LIN {X 0,Y 254.112,Z 618.126,A -85,B 0,C 180,E1 -18637.149,E2 -18637.149} C_VEL
LIN {X 0,Y 253.777,Z 620.989,A -85,B 0,C 180,E1 -18639.564,E2 -18639.564} C_VEL
LIN {X 0,Y 253.688,Z 622.339,A -85,B 0,C 180,E1 -18641.181,E2 -18641.181} C_VEL
LIN {X 0,Y 253.728,Z 623.768,A -85,B 0,C 180,E1 -18644.196,E2 -18644.196} C_VEL
LIN {X 0,Y 253.789,Z 623.911,A -85,B 0,C 180,E1 -18646.076,E2 -18646.076} C_VEL
LIN {X 0,Y 253.947,Z 623.596,A -85,B 0,C 180,E1 -18647.723,E2 -18647.723} C_VEL
LIN {X 0,Y 254.457,Z 622.389,A -85,B 0,C 180,E1 -18650.104,E2 -18650.104} C_VEL
LIN {X 0,Y 255.585,Z 619.098,A -85,B 0,C 180,E1 -18653.497,E2 -18653.497} C_VEL
LIN {X 0,Y 256.833,Z 615.411,A -85,B 0,C 180,E1 -18655.964,E2 -18655.964} C_VEL
LIN {X 0,Y 258.431,Z 610.517,A -85,B 0,C 180,E1 -18658.418,E2 -18658.418} C_VEL
LIN {X 0,Y 260.518,Z 604.271,A -85,B 0,C 180,E1 -18660.834,E2 -18660.834} C_VEL
LIN {X 0,Y 262.965,Z 596.427,A -85,B 0,C 180,E1 -18663.221,E2 -18663.221} C_VEL
LIN {X 0,Y 265.473,Z 587.888,A -85,B 0,C 180,E1 -18665.261,E2 -18665.261} C_VEL
LIN {X 0,Y 268.117,Z 578.332,A -85,B 0,C 180,E1 -18667.076,E2 -18667.076} C_VEL
LIN {X 0,Y 270.488,Z 568.5,A -85,B 0,C 180,E1 -18668.577,E2 -18668.577} C_VEL
LIN {X 0,Y 272.671,Z 557.853,A -85,B 0,C 180,E1 -18669.877,E2 -18669.877} C_VEL
LIN {X 0,Y 274.602,Z 546.18,A -85,B 0,C 180,E1 -18670.981,E2 -18670.981} C_VEL
LIN {X 0,Y 276.337,Z 533.273,A -85,B 0,C 180,E1 -18671.853,E2 -18671.853} C_VEL
LIN {X 0,Y 277.554,Z 520.336,A -85,B 0,C 180,E1 -18672.432,E2 -18672.432} C_VEL
LIN {X 0,Y 280.067,Z 457.156,A -85,B 0,C 180,E1 -18674.084,E2 -18674.084} C_VEL
LIN {X 0,Y 274.463,Z 444.134,A -85,B 0,C 180,E1 -18675.366,E2 -18675.366} C_VEL
LIN {X 0,Y 267.207,Z 429.8,A -85,B 0,C 180,E1 -18677.057,E2 -18677.057} C_VEL
LIN {X 0,Y 260.209,Z 417.558,A -85,B 0,C 180,E1 -18678.762,E2 -18678.762} C_VEL
LIN {X 0,Y 257.879,Z 413.399,A -85,B 0,C 180,E1 -18679.453,E2 -18679.453} C_VEL
LIN {X 0,Y 256.173,Z 407.244,A -85,B 0,C 180,E1 -18682.71,E2 -18682.71} C_VEL
LIN {X 0,Y 256.081,Z 407.076,A -85,B 0,C 180,E1 -18686.709,E2 -18686.709} C_VEL
LIN {X 0,Y 256.122,Z 407.062,A -85,B 0,C 180,E1 -18691.409,E2 -18691.409} C_VEL
LIN {X 0,Y 256.162,Z 407.076,A -85,B 0,C 180,E1 -18695.699,E2 -18695.699} C_VEL
LIN {X 0,Y 256.162,Z 407.074,A -85,B 0,C 180,E1 -18699.105,E2 -18699.105} C_VEL
LIN {X 0,Y 256.289,Z 407.06,A -85,B 0,C 180,E1 -18704.084,E2 -18704.084} C_VEL
LIN {X 0,Y 256.304,Z 407.05,A -85,B 0,C 180,E1 -18708.934,E2 -18708.934} C_VEL
LIN {X 0,Y 256.533,Z 407.03,A -85,B 0,C 180,E1 -18712.127,E2 -18712.127} C_VEL
LIN {X 0,Y 256.347,Z 407.044,A -85,B 0,C 180,E1 -18715.171,E2 -18715.171} C_VEL
LIN {X 0,Y 255.716,Z 407.133,A -85,B 0,C 180,E1 -18716.486,E2 -18716.486} C_VEL
LIN {X 0,Y 253.085,Z 407.469,A -85,B 0,C 180,E1 -18718.637,E2 -18718.637} C_VEL
LIN {X 0,Y 249.973,Z 407.849,A -85,B 0,C 180,E1 -18721.28,E2 -18721.28} C_VEL
LIN {X 0,Y 249.565,Z 407.891,A -85,B 0,C 180,E1 -18722.191,E2 -18722.191} C_VEL
LIN {X 0,Y 249.455,Z 407.913,A -85,B 0,C 180,E1 -18726.471,E2 -18726.471} C_VEL
LIN {X 0,Y 249.383,Z 407.911,A -85,B 0,C 180,E1 -18729.735,E2 -18729.735} C_VEL
LIN {X 0,Y 249.199,Z 407.934,A -85,B 0,C 180,E1 -18734.704,E2 -18734.704} C_VEL
LIN {X 0,Y 249.134,Z 407.939,A -85,B 0,C 180,E1 -18738.078,E2 -18738.078} C_VEL
LIN {X 0,Y 249.082,Z 407.953,A -85,B 0,C 180,E1 -18741.519,E2 -18741.519} C_VEL
LIN {X 0,Y 249.126,Z 407.95,A -85,B 0,C 180,E1 -18745.483,E2 -18745.483} C_VEL
LIN {X 0,Y 249.079,Z 407.959,A -85,B 0,C 180,E1 -18748.994,E2 -18748.994} C_VEL
LIN {X 0,Y 249.032,Z 407.966,A -85,B 0,C 180,E1 -18752.426,E2 -18752.426} C_VEL
LIN {X 0,Y 249.072,Z 407.958,A -85,B 0,C 180,E1 -18756.339,E2 -18756.339} C_VEL
LIN {X 0,Y 249.082,Z 407.938,A -85,B 0,C 180,E1 -18760.463,E2 -18760.463} C_VEL
LIN {X 0,Y 249.017,Z 407.957,A -85,B 0,C 180,E1 -18764.876,E2 -18764.876} C_VEL
LIN {X 0,Y 249.039,Z 407.996,A -85,B 0,C 180,E1 -18766.648,E2 -18766.648} C_VEL
LIN {X 0,Y 250.574,Z 413.471,A -85,B 0,C 180,E1 -18769.829,E2 -18769.829} C_VEL
LIN {X 0,Y 252.023,Z 418.69,A -85,B 0,C 180,E1 -18772.439,E2 -18772.439} C_VEL
LIN {X 0,Y 254.643,Z 423.279,A -85,B 0,C 180,E1 -18773.215,E2 -18773.215} C_VEL
LIN {X 0,Y 263.1,Z 438.828,A -85,B 0,C 180,E1 -18775.383,E2 -18775.383} C_VEL
LIN {X 0,Y 270.526,Z 454.405,A -85,B 0,C 180,E1 -18777.189,E2 -18777.189} C_VEL
LIN {X 0,Y 272.23,Z 459.018,A -85,B 0,C 180,E1 -18777.618,E2 -18777.618} C_VEL
LIN {X 0,Y 273.963,Z 469.57,A -85,B 0,C 180,E1 -18778.237,E2 -18778.237} C_VEL
LIN {X 0,Y 271.409,Z 527.607,A -85,B 0,C 180,E1 -18779.779,E2 -18779.779} C_VEL
LIN {X 0,Y 270.097,Z 541.162,A -85,B 0,C 180,E1 -18780.425,E2 -18780.425} C_VEL
LIN {X 0,Y 268.197,Z 553.913,A -85,B 0,C 180,E1 -18781.324,E2 -18781.324} C_VEL
LIN {X 0,Y 265.918,Z 565.575,A -85,B 0,C 180,E1 -18782.452,E2 -18782.452} C_VEL
LIN {X 0,Y 263.435,Z 576.821,A -85,B 0,C 180,E1 -18783.885,E2 -18783.885} C_VEL
LIN {X 0,Y 260.778,Z 586.995,A -85,B 0,C 180,E1 -18785.522,E2 -18785.522} C_VEL
LIN {X 0,Y 257.805,Z 596.965,A -85,B 0,C 180,E1 -18787.565,E2 -18787.565} C_VEL
LIN {X 0,Y 255.094,Z 605.859,A -85,B 0,C 180,E1 -18789.894,E2 -18789.894} C_VEL
LIN {X 0,Y 252.844,Z 612.807,A -85,B 0,C 180,E1 -18792.197,E2 -18792.197} C_VEL
LIN {X 0,Y 250.801,Z 618.469,A -85,B 0,C 180,E1 -18794.562,E2 -18794.562} C_VEL
LIN {X 0,Y 249.326,Z 622.943,A -85,B 0,C 180,E1 -18796.968,E2 -18796.968} C_VEL
LIN {X 0,Y 248.525,Z 625.31,A -85,B 0,C 180,E1 -18798.583,E2 -18798.583} C_VEL
LIN {X 0,Y 247.412,Z 628.797,A -85,B 0,C 180,E1 -18801.835,E2 -18801.835} C_VEL
LIN {X 0,Y 246.945,Z 630.557,A -85,B 0,C 180,E1 -18804.937,E2 -18804.937} C_VEL
LIN {X 0,Y 246.831,Z 630.932,A -85,B 0,C 180,E1 -18806.736,E2 -18806.736} C_VEL
LIN {X 0,Y 246.859,Z 630.877,A -85,B 0,C 180,E1 -18808.369,E2 -18808.369} C_VEL
LIN {X 0,Y 246.899,Z 630.414,A -85,B 0,C 180,E1 -18810,E2 -18810} C_VEL
LIN {X 0,Y 246.86,Z 629.526,A -85,B 0,C 180,E1 -18811.632,E2 -18811.632} C_VEL
LIN {X 0,Y 246.831,Z 628.24,A -85,B 0,C 180,E1 -18813.265,E2 -18813.265} C_VEL
LIN {X 0,Y 246.906,Z 625.502,A -85,B 0,C 180,E1 -18815.718,E2 -18815.718} C_VEL
LIN {X 0,Y 247.269,Z 621.729,A -85,B 0,C 180,E1 -18818.17,E2 -18818.17} C_VEL
LIN {X 0,Y 247.852,Z 616.812,A -85,B 0,C 180,E1 -18820.621,E2 -18820.621} C_VEL
LIN {X 0,Y 248.729,Z 610.599,A -85,B 0,C 180,E1 -18823.064,E2 -18823.064} C_VEL
LIN {X 0,Y 250.11,Z 602.853,A -85,B 0,C 180,E1 -18825.483,E2 -18825.483} C_VEL
LIN {X 0,Y 251.484,Z 594.894,A -85,B 0,C 180,E1 -18827.483,E2 -18827.483} C_VEL
LIN {X 0,Y 252.89,Z 585.135,A -85,B 0,C 180,E1 -18829.481,E2 -18829.481} C_VEL
LIN {X 0,Y 254.533,Z 574.299,A -85,B 0,C 180,E1 -18831.248,E2 -18831.248} C_VEL
LIN {X 0,Y 256.086,Z 563.781,A -85,B 0,C 180,E1 -18832.595,E2 -18832.595} C_VEL
LIN {X 0,Y 257.649,Z 551.092,A -85,B 0,C 180,E1 -18833.831,E2 -18833.831} C_VEL
LIN {X 0,Y 258.828,Z 537.613,A -85,B 0,C 180,E1 -18834.782,E2 -18834.782} C_VEL
LIN {X 0,Y 259.618,Z 525.011,A -85,B 0,C 180,E1 -18835.344,E2 -18835.344} C_VEL
LIN {X 0,Y 261.246,Z 462.897,A -85,B 0,C 180,E1 -18837.047,E2 -18837.047} C_VEL
LIN {X 0,Y 257.5,Z 435.906,A -85,B 0,C 180,E1 -18838.198,E2 -18838.198} C_VEL
LIN {X 0,Y 251.549,Z 419.268,A -85,B 0,C 180,E1 -18839.345,E2 -18839.345} C_VEL
LIN {X 0,Y 249.312,Z 409.016,A -85,B 0,C 180,E1 -18843.345,E2 -18843.345} C_VEL
LIN {X 0,Y 249.092,Z 407.982,A -85,B 0,C 180,E1 -18843.925,E2 -18843.925} C_VEL
LIN {X 0,Y 249.043,Z 407.95,A -85,B 0,C 180,E1 -18848.377,E2 -18848.377} C_VEL
LIN {X 0,Y 249.044,Z 407.961,A -85,B 0,C 180,E1 -18852.801,E2 -18852.801} C_VEL
LIN {X 0,Y 249.062,Z 407.934,A -85,B 0,C 180,E1 -18857.372,E2 -18857.372} C_VEL
LIN {X 0,Y 249.052,Z 407.962,A -85,B 0,C 180,E1 -18861.624,E2 -18861.624} C_VEL
LIN {X 0,Y 249.061,Z 407.957,A -85,B 0,C 180,E1 -18865.642,E2 -18865.642} C_VEL
LIN {X 0,Y 249.046,Z 407.957,A -85,B 0,C 180,E1 -18869.472,E2 -18869.472} C_VEL
LIN {X 0,Y 249.067,Z 407.954,A -85,B 0,C 180,E1 -18873.161,E2 -18873.161} C_VEL
LIN {X 0,Y 249.059,Z 407.959,A -85,B 0,C 180,E1 -18876.73,E2 -18876.73} C_VEL
LIN {X 0,Y 249.105,Z 407.938,A -85,B 0,C 180,E1 -18880.211,E2 -18880.211} C_VEL
LIN {X 0,Y 249.24,Z 407.939,A -85,B 0,C 180,E1 -18883.622,E2 -18883.622} C_VEL
LIN {X 0,Y 249.241,Z 407.922,A -85,B 0,C 180,E1 -18888.616,E2 -18888.616} C_VEL
LIN {X 0,Y 249.452,Z 407.904,A -85,B 0,C 180,E1 -18891.902,E2 -18891.902} C_VEL
LIN {X 0,Y 249.294,Z 407.933,A -85,B 0,C 180,E1 -18895.148,E2 -18895.148} C_VEL
LIN {X 0,Y 249.673,Z 407.875,A -85,B 0,C 180,E1 -18898.387,E2 -18898.387} C_VEL
LIN {X 0,Y 249.673,Z 407.862,A -85,B 0,C 180,E1 -18901.613,E2 -18901.613} C_VEL
LIN {X 0,Y 249.438,Z 407.91,A -85,B 0,C 180,E1 -18906.711,E2 -18906.711} C_VEL
LIN {X 0,Y 249.341,Z 407.915,A -85,B 0,C 180,E1 -18909.736,E2 -18909.736} C_VEL
LIN {X 0,Y 249.198,Z 407.93,A -85,B 0,C 180,E1 -18914.704,E2 -18914.704} C_VEL
LIN {X 0,Y 249.136,Z 407.949,A -85,B 0,C 180,E1 -18918.077,E2 -18918.077} C_VEL
LIN {X 0,Y 249.085,Z 407.945,A -85,B 0,C 180,E1 -18921.518,E2 -18921.518} C_VEL
LIN {X 0,Y 249.128,Z 407.939,A -85,B 0,C 180,E1 -18925.482,E2 -18925.482} C_VEL
LIN {X 0,Y 249.081,Z 407.958,A -85,B 0,C 180,E1 -18928.993,E2 -18928.993} C_VEL
LIN {X 0,Y 249.028,Z 407.952,A -85,B 0,C 180,E1 -18932.426,E2 -18932.426} C_VEL
LIN {X 0,Y 249.046,Z 407.957,A -85,B 0,C 180,E1 -18936.343,E2 -18936.343} C_VEL
LIN {X 0,Y 249.004,Z 407.963,A -85,B 0,C 180,E1 -18940.478,E2 -18940.478} C_VEL
LIN {X 0,Y 249.009,Z 407.966,A -85,B 0,C 180,E1 -18944.878,E2 -18944.878} C_VEL
LIN {X 0,Y 249.036,Z 407.96,A -85,B 0,C 180,E1 -18947.368,E2 -18947.368} C_VEL
LIN {X 0,Y 249.051,Z 407.964,A -85,B 0,C 180,E1 -18951.624,E2 -18951.624} C_VEL
LIN {X 0,Y 249.061,Z 407.942,A -85,B 0,C 180,E1 -18955.643,E2 -18955.643} C_VEL
LIN {X 0,Y 249.052,Z 407.947,A -85,B 0,C 180,E1 -18959.473,E2 -18959.473} C_VEL
LIN {X 0,Y 249.074,Z 407.951,A -85,B 0,C 180,E1 -18963.162,E2 -18963.162} C_VEL
LIN {X 0,Y 249.08,Z 407.948,A -85,B 0,C 180,E1 -18966.733,E2 -18966.733} C_VEL
LIN {X 0,Y 249.196,Z 408.095,A -85,B 0,C 180,E1 -18971.555,E2 -18971.555} C_VEL
LIN {X 0,Y 250.291,Z 413.05,A -85,B 0,C 180,E1 -18973.576,E2 -18973.576} C_VEL
LIN {X 0,Y 256.255,Z 428.663,A -85,B 0,C 180,E1 -18974.719,E2 -18974.719} C_VEL
LIN {X 0,Y 259.336,Z 438.01,A -85,B 0,C 180,E1 -18975.295,E2 -18975.295} C_VEL
LIN {X 0,Y 261.649,Z 453.277,A -85,B 0,C 180,E1 -18975.961,E2 -18975.961} C_VEL
LIN {X 0,Y 259.555,Z 520.29,A -85,B 0,C 180,E1 -18977.787,E2 -18977.787} C_VEL
LIN {X 0,Y 258.768,Z 533.398,A -85,B 0,C 180,E1 -18978.445,E2 -18978.445} C_VEL
LIN {X 0,Y 257.68,Z 545.229,A -85,B 0,C 180,E1 -18979.316,E2 -18979.316} C_VEL
LIN {X 0,Y 256.248,Z 557.373,A -85,B 0,C 180,E1 -18980.528,E2 -18980.528} C_VEL
LIN {X 0,Y 254.517,Z 569.044,A -85,B 0,C 180,E1 -18982.064,E2 -18982.064} C_VEL
LIN {X 0,Y 253.082,Z 578.437,A -85,B 0,C 180,E1 -18983.622,E2 -18983.622} C_VEL
LIN {X 0,Y 251.443,Z 588.078,A -85,B 0,C 180,E1 -18985.591,E2 -18985.591} C_VEL
LIN {X 0,Y 250.22,Z 595.954,A -85,B 0,C 180,E1 -18987.585,E2 -18987.585} C_VEL
LIN {X 0,Y 248.882,Z 603.666,A -85,B 0,C 180,E1 -18990,E2 -18990} C_VEL
LIN {X 0,Y 247.955,Z 609.852,A -85,B 0,C 180,E1 -18992.436,E2 -18992.436} C_VEL
LIN {X 0,Y 247.399,Z 614.759,A -85,B 0,C 180,E1 -18994.888,E2 -18994.888} C_VEL
LIN {X 0,Y 246.973,Z 618.549,A -85,B 0,C 180,E1 -18997.357,E2 -18997.357} C_VEL
LIN {X 0,Y 246.675,Z 621.31,A -85,B 0,C 180,E1 -18999.842,E2 -18999.842} C_VEL
LIN {X 0,Y 246.598,Z 622.611,A -85,B 0,C 180,E1 -19001.507,E2 -19001.507} C_VEL
LIN {X 0,Y 246.648,Z 623.865,A -85,B 0,C 180,E1 -19004.35,E2 -19004.35} C_VEL
LIN {X 0,Y 246.737,Z 623.989,A -85,B 0,C 180,E1 -19006.548,E2 -19006.548} C_VEL
LIN {X 0,Y 246.954,Z 623.626,A -85,B 0,C 180,E1 -19008.242,E2 -19008.242} C_VEL
LIN {X 0,Y 247.432,Z 622.525,A -85,B 0,C 180,E1 -19010.393,E2 -19010.393} C_VEL
LIN {X 0,Y 248.394,Z 619.898,A -85,B 0,C 180,E1 -19013.334,E2 -19013.334} C_VEL
LIN {X 0,Y 249.537,Z 616.773,A -85,B 0,C 180,E1 -19015.677,E2 -19015.677} C_VEL
LIN {X 0,Y 251.248,Z 611.893,A -85,B 0,C 180,E1 -19018.393,E2 -19018.393} C_VEL
LIN {X 0,Y 253.528,Z 605.511,A -85,B 0,C 180,E1 -19021.049,E2 -19021.049} C_VEL
LIN {X 0,Y 255.822,Z 598.512,A -85,B 0,C 180,E1 -19023.328,E2 -19023.328} C_VEL
LIN {X 0,Y 258.479,Z 590.1,A -85,B 0,C 180,E1 -19025.502,E2 -19025.502} C_VEL
LIN {X 0,Y 261.351,Z 580.456,A -85,B 0,C 180,E1 -19027.473,E2 -19027.473} C_VEL
LIN {X 0,Y 264.095,Z 569.707,A -85,B 0,C 180,E1 -19029.198,E2 -19029.198} C_VEL
LIN {X 0,Y 266.618,Z 558.006,A -85,B 0,C 180,E1 -19030.672,E2 -19030.672} C_VEL
LIN {X 0,Y 268.715,Z 545.893,A -85,B 0,C 180,E1 -19031.829,E2 -19031.829} C_VEL
LIN {X 0,Y 270.575,Z 532.505,A -85,B 0,C 180,E1 -19032.731,E2 -19032.731} C_VEL
LIN {X 0,Y 271.77,Z 519.507,A -85,B 0,C 180,E1 -19033.307,E2 -19033.307} C_VEL
LIN {X 0,Y 274.325,Z 459.31,A -85,B 0,C 180,E1 -19034.892,E2 -19034.892} C_VEL
LIN {X 0,Y 268.112,Z 445.144,A -85,B 0,C 180,E1 -19036.376,E2 -19036.376} C_VEL
LIN {X 0,Y 260.809,Z 430.871,A -85,B 0,C 180,E1 -19038.169,E2 -19038.169} C_VEL
LIN {X 0,Y 253.015,Z 417.7,A -85,B 0,C 180,E1 -19040.177,E2 -19040.177} C_VEL
LIN {X 0,Y 250.681,Z 413.682,A -85,B 0,C 180,E1 -19040.891,E2 -19040.891} C_VEL
LIN {X 0,Y 249.687,Z 410.098,A -85,B 0,C 180,E1 -19042.759,E2 -19042.759} C_VEL
LIN {X 0,Y 249.091,Z 407.978,A -85,B 0,C 180,E1 -19044.145,E2 -19044.145} C_VEL
LIN {X 0,Y 249.035,Z 407.965,A -85,B 0,C 180,E1 -19047.844,E2 -19047.844} C_VEL
LIN {X 0,Y 249.081,Z 407.938,A -85,B 0,C 180,E1 -19051.336,E2 -19051.336} C_VEL
LIN {X 0,Y 249.147,Z 407.945,A -85,B 0,C 180,E1 -19054.968,E2 -19054.968} C_VEL
LIN {X 0,Y 249.106,Z 407.955,A -85,B 0,C 180,E1 -19060.211,E2 -19060.211} C_VEL
LIN {X 0,Y 249.236,Z 407.939,A -85,B 0,C 180,E1 -19063.622,E2 -19063.622} C_VEL
LIN {X 0,Y 249.247,Z 407.932,A -85,B 0,C 180,E1 -19068.616,E2 -19068.616} C_VEL
LIN {X 0,Y 249.475,Z 407.909,A -85,B 0,C 180,E1 -19071.903,E2 -19071.903} C_VEL
LIN {X 0,Y 249.462,Z 407.913,A -85,B 0,C 180,E1 -19076.77,E2 -19076.77} C_VEL
LIN {X 0,Y 249.73,Z 407.868,A -85,B 0,C 180,E1 -19080,E2 -19080} C_VEL
LIN {X 0,Y 249.565,Z 407.891,A -85,B 0,C 180,E1 -19082.191,E2 -19082.191} C_VEL
LIN {X 0,Y 248.748,Z 407.989,A -85,B 0,C 180,E1 -19083.537,E2 -19083.537} C_VEL
LIN {X 0,Y 245.844,Z 408.361,A -85,B 0,C 180,E1 -19085.733,E2 -19085.733} C_VEL
LIN {X 0,Y 243.465,Z 408.652,A -85,B 0,C 180,E1 -19087.521,E2 -19087.521} C_VEL
LIN {X 0,Y 242.448,Z 408.771,A -85,B 0,C 180,E1 -19088.907,E2 -19088.907} C_VEL
LIN {X 0,Y 242.362,Z 408.783,A -85,B 0,C 180,E1 -19089.377,E2 -19089.377} C_VEL
LIN {X 0,Y 242.161,Z 408.815,A -85,B 0,C 180,E1 -19095.141,E2 -19095.141} C_VEL
LIN {X 0,Y 242.068,Z 408.819,A -85,B 0,C 180,E1 -19098.625,E2 -19098.625} C_VEL
LIN {X 0,Y 242.008,Z 408.829,A -85,B 0,C 180,E1 -19102.181,E2 -19102.181} C_VEL
LIN {X 0,Y 242.062,Z 408.826,A -85,B 0,C 180,E1 -19105.839,E2 -19105.839} C_VEL
LIN {X 0,Y 242.026,Z 408.834,A -85,B 0,C 180,E1 -19109.581,E2 -19109.581} C_VEL
LIN {X 0,Y 241.987,Z 408.836,A -85,B 0,C 180,E1 -19113.492,E2 -19113.492} C_VEL
LIN {X 0,Y 242.016,Z 408.832,A -85,B 0,C 180,E1 -19117.577,E2 -19117.577} C_VEL
LIN {X 0,Y 241.984,Z 408.817,A -85,B 0,C 180,E1 -19121.913,E2 -19121.913} C_VEL
LIN {X 0,Y 241.995,Z 409.041,A -85,B 0,C 180,E1 -19125.45,E2 -19125.45} C_VEL
LIN {X 0,Y 244.075,Z 416.279,A -85,B 0,C 180,E1 -19129.717,E2 -19129.717} C_VEL
LIN {X 0,Y 244.789,Z 418.663,A -85,B 0,C 180,E1 -19130.877,E2 -19130.877} C_VEL
LIN {X 0,Y 247.405,Z 423.195,A -85,B 0,C 180,E1 -19131.703,E2 -19131.703} C_VEL
LIN {X 0,Y 253.58,Z 434.009,A -85,B 0,C 180,E1 -19133.406,E2 -19133.406} C_VEL
LIN {X 0,Y 259.89,Z 446.068,A -85,B 0,C 180,E1 -19135.057,E2 -19135.057} C_VEL
LIN {X 0,Y 266.039,Z 459.536,A -85,B 0,C 180,E1 -19136.615,E2 -19136.615} C_VEL
LIN {X 0,Y 266.95,Z 462.519,A -85,B 0,C 180,E1 -19136.87,E2 -19136.87} C_VEL
LIN {X 0,Y 268.284,Z 470.283,A -85,B 0,C 180,E1 -19137.354,E2 -19137.354} C_VEL
LIN {X 0,Y 265.717,Z 526.862,A -85,B 0,C 180,E1 -19138.878,E2 -19138.878} C_VEL
LIN {X 0,Y 264.317,Z 540.529,A -85,B 0,C 180,E1 -19139.52,E2 -19139.52} C_VEL
LIN {X 0,Y 262.427,Z 553.183,A -85,B 0,C 180,E1 -19140.412,E2 -19140.412} C_VEL
LIN {X 0,Y 260.04,Z 564.991,A -85,B 0,C 180,E1 -19141.554,E2 -19141.554} C_VEL
LIN {X 0,Y 257.463,Z 576.317,A -85,B 0,C 180,E1 -19143.012,E2 -19143.012} C_VEL
LIN {X 0,Y 254.697,Z 586.561,A -85,B 0,C 180,E1 -19144.679,E2 -19144.679} C_VEL
LIN {X 0,Y 251.817,Z 595.795,A -85,B 0,C 180,E1 -19146.566,E2 -19146.566} C_VEL
LIN {X 0,Y 249.014,Z 604.498,A -85,B 0,C 180,E1 -19148.831,E2 -19148.831} C_VEL
LIN {X 0,Y 246.517,Z 611.976,A -85,B 0,C 180,E1 -19151.294,E2 -19151.294} C_VEL
LIN {X 0,Y 244.613,Z 616.899,A -85,B 0,C 180,E1 -19153.304,E2 -19153.304} C_VEL
LIN {X 0,Y 242.857,Z 621.69,A -85,B 0,C 180,E1 -19155.761,E2 -19155.761} C_VEL
LIN {X 0,Y 241.554,Z 625.386,A -85,B 0,C 180,E1 -19158.249,E2 -19158.249} C_VEL
LIN {X 0,Y 240.891,Z 627.303,A -85,B 0,C 180,E1 -19159.919,E2 -19159.919} C_VEL
LIN {X 0,Y 240.386,Z 628.805,A -85,B 0,C 180,E1 -19161.595,E2 -19161.595} C_VEL
LIN {X 0,Y 239.845,Z 630.545,A -85,B 0,C 180,E1 -19164.957,E2 -19164.957} C_VEL
LIN {X 0,Y 239.773,Z 630.76,A -85,B 0,C 180,E1 -19168.321,E2 -19168.321} C_VEL
LIN {X 0,Y 239.811,Z 630.247,A -85,B 0,C 180,E1 -19170,E2 -19170} C_VEL
LIN {X 0,Y 239.774,Z 629.332,A -85,B 0,C 180,E1 -19171.68,E2 -19171.68} C_VEL
LIN {X 0,Y 239.766,Z 626.645,A -85,B 0,C 180,E1 -19174.718,E2 -19174.718} C_VEL
LIN {X 0,Y 240.048,Z 622.813,A -85,B 0,C 180,E1 -19177.571,E2 -19177.571} C_VEL
LIN {X 0,Y 240.618,Z 618.229,A -85,B 0,C 180,E1 -19180.093,E2 -19180.093} C_VEL
LIN {X 0,Y 241.584,Z 611.251,A -85,B 0,C 180,E1 -19183.03,E2 -19183.03} C_VEL
LIN {X 0,Y 242.966,Z 603.689,A -85,B 0,C 180,E1 -19185.519,E2 -19185.519} C_VEL
LIN {X 0,Y 244.362,Z 595.951,A -85,B 0,C 180,E1 -19187.577,E2 -19187.577} C_VEL
LIN {X 0,Y 245.888,Z 586.075,A -85,B 0,C 180,E1 -19189.705,E2 -19189.705} C_VEL
LIN {X 0,Y 247.671,Z 574.634,A -85,B 0,C 180,E1 -19191.647,E2 -19191.647} C_VEL
LIN {X 0,Y 249.272,Z 564.232,A -85,B 0,C 180,E1 -19193.029,E2 -19193.029} C_VEL
LIN {X 0,Y 250.871,Z 551.751,A -85,B 0,C 180,E1 -19194.297,E2 -19194.297} C_VEL
LIN {X 0,Y 252.104,Z 538.553,A -85,B 0,C 180,E1 -19195.269,E2 -19195.269} C_VEL
LIN {X 0,Y 252.968,Z 525.413,A -85,B 0,C 180,E1 -19195.893,E2 -19195.893} C_VEL
LIN {X 0,Y 254.789,Z 464.792,A -85,B 0,C 180,E1 -19197.584,E2 -19197.584} C_VEL
LIN {X 0,Y 251.148,Z 438.097,A -85,B 0,C 180,E1 -19198.758,E2 -19198.758} C_VEL
LIN {X 0,Y 245.146,Z 421.605,A -85,B 0,C 180,E1 -19199.902,E2 -19199.902} C_VEL
LIN {X 0,Y 244.224,Z 418.953,A -85,B 0,C 180,E1 -19200.175,E2 -19200.175} C_VEL
LIN {X 0,Y 242.201,Z 409.661,A -85,B 0,C 180,E1 -19203.957,E2 -19203.957} C_VEL
LIN {X 0,Y 242.042,Z 408.85,A -85,B 0,C 180,E1 -19204.486,E2 -19204.486} C_VEL
LIN {X 0,Y 242.011,Z 408.825,A -85,B 0,C 180,E1 -19208.364,E2 -19208.364} C_VEL
LIN {X 0,Y 241.966,Z 408.845,A -85,B 0,C 180,E1 -19211.916,E2 -19211.916} C_VEL
LIN {X 0,Y 241.991,Z 408.807,A -85,B 0,C 180,E1 -19216.557,E2 -19216.557} C_VEL
LIN {X 0,Y 242.008,Z 408.839,A -85,B 0,C 180,E1 -19220.291,E2 -19220.291} C_VEL
LIN {X 0,Y 242.036,Z 408.825,A -85,B 0,C 180,E1 -19224.497,E2 -19224.497} C_VEL
LIN {X 0,Y 241.973,Z 408.843,A -85,B 0,C 180,E1 -19228.479,E2 -19228.479} C_VEL
LIN {X 0,Y 241.999,Z 408.831,A -85,B 0,C 180,E1 -19232.311,E2 -19232.311} C_VEL
LIN {X 0,Y 242.039,Z 408.834,A -85,B 0,C 180,E1 -19236.014,E2 -19236.014} C_VEL
LIN {X 0,Y 242.033,Z 408.817,A -85,B 0,C 180,E1 -19239.607,E2 -19239.607} C_VEL
LIN {X 0,Y 242.161,Z 408.818,A -85,B 0,C 180,E1 -19243.278,E2 -19243.278} C_VEL
LIN {X 0,Y 242.178,Z 408.803,A -85,B 0,C 180,E1 -19248.279,E2 -19248.279} C_VEL
LIN {X 0,Y 242.398,Z 408.778,A -85,B 0,C 180,E1 -19251.664,E2 -19251.664} C_VEL
LIN {X 0,Y 242.255,Z 408.809,A -85,B 0,C 180,E1 -19255.007,E2 -19255.007} C_VEL
LIN {X 0,Y 242.633,Z 408.752,A -85,B 0,C 180,E1 -19258.34,E2 -19258.34} C_VEL
LIN {X 0,Y 242.633,Z 408.738,A -85,B 0,C 180,E1 -19261.66,E2 -19261.66} C_VEL
LIN {X 0,Y 242.419,Z 408.787,A -85,B 0,C 180,E1 -19266.683,E2 -19266.683} C_VEL
LIN {X 0,Y 242.265,Z 408.795,A -85,B 0,C 180,E1 -19270.024,E2 -19270.024} C_VEL
LIN {X 0,Y 242.161,Z 408.809,A -85,B 0,C 180,E1 -19275.141,E2 -19275.141} C_VEL
LIN {X 0,Y 242.07,Z 408.83,A -85,B 0,C 180,E1 -19278.624,E2 -19278.624} C_VEL
LIN {X 0,Y 242.011,Z 408.824,A -85,B 0,C 180,E1 -19282.18,E2 -19282.18} C_VEL
LIN {X 0,Y 242.065,Z 408.822,A -85,B 0,C 180,E1 -19285.838,E2 -19285.838} C_VEL
LIN {X 0,Y 242.028,Z 408.834,A -85,B 0,C 180,E1 -19289.58,E2 -19289.58} C_VEL
LIN {X 0,Y 241.979,Z 408.823,A -85,B 0,C 180,E1 -19293.493,E2 -19293.493} C_VEL
LIN {X 0,Y 241.987,Z 408.842,A -85,B 0,C 180,E1 -19297.582,E2 -19297.582} C_VEL
LIN {X 0,Y 241.938,Z 408.83,A -85,B 0,C 180,E1 -19301.922,E2 -19301.922} C_VEL
LIN {X 0,Y 241.973,Z 408.844,A -85,B 0,C 180,E1 -19306.561,E2 -19306.561} C_VEL
LIN {X 0,Y 241.987,Z 408.837,A -85,B 0,C 180,E1 -19310.287,E2 -19310.287} C_VEL
LIN {X 0,Y 242.037,Z 408.826,A -85,B 0,C 180,E1 -19314.498,E2 -19314.498} C_VEL
LIN {X 0,Y 241.976,Z 408.814,A -85,B 0,C 180,E1 -19318.48,E2 -19318.48} C_VEL
LIN {X 0,Y 242.01,Z 408.839,A -85,B 0,C 180,E1 -19322.313,E2 -19322.313} C_VEL
LIN {X 0,Y 242.058,Z 408.812,A -85,B 0,C 180,E1 -19326.016,E2 -19326.016} C_VEL
LIN {X 0,Y 242.174,Z 408.986,A -85,B 0,C 180,E1 -19331.055,E2 -19331.055} C_VEL
LIN {X 0,Y 243.104,Z 413.283,A -85,B 0,C 180,E1 -19332.812,E2 -19332.812} C_VEL
LIN {X 0,Y 249.796,Z 430.382,A -85,B 0,C 180,E1 -19334.12,E2 -19334.12} C_VEL
LIN {X 0,Y 253.035,Z 440.431,A -85,B 0,C 180,E1 -19334.758,E2 -19334.758} C_VEL
LIN {X 0,Y 255.082,Z 454.542,A -85,B 0,C 180,E1 -19335.388,E2 -19335.388} C_VEL
LIN {X 0,Y 252.96,Z 520.007,A -85,B 0,C 180,E1 -19337.209,E2 -19337.209} C_VEL
LIN {X 0,Y 252.117,Z 533.257,A -85,B 0,C 180,E1 -19337.881,E2 -19337.881} C_VEL
LIN {X 0,Y 250.877,Z 546.548,A -85,B 0,C 180,E1 -19338.895,E2 -19338.895} C_VEL
LIN {X 0,Y 249.469,Z 557.738,A -85,B 0,C 180,E1 -19340.063,E2 -19340.063} C_VEL
LIN {X 0,Y 247.68,Z 569.362,A -85,B 0,C 180,E1 -19341.638,E2 -19341.638} C_VEL
LIN {X 0,Y 246.199,Z 578.717,A -85,B 0,C 180,E1 -19343.237,E2 -19343.237} C_VEL
LIN {X 0,Y 244.675,Z 587.432,A -85,B 0,C 180,E1 -19345.056,E2 -19345.056} C_VEL
LIN {X 0,Y 243.355,Z 595.435,A -85,B 0,C 180,E1 -19347.103,E2 -19347.103} C_VEL
LIN {X 0,Y 241.931,Z 603.301,A -85,B 0,C 180,E1 -19349.583,E2 -19349.583} C_VEL
LIN {X 0,Y 241.163,Z 608.631,A -85,B 0,C 180,E1 -19351.67,E2 -19351.67} C_VEL
LIN {X 0,Y 240.45,Z 613.833,A -85,B 0,C 180,E1 -19354.19,E2 -19354.19} C_VEL
LIN {X 0,Y 239.989,Z 617.877,A -85,B 0,C 180,E1 -19356.726,E2 -19356.726} C_VEL
LIN {X 0,Y 239.691,Z 619.967,A -85,B 0,C 180,E1 -19358.43,E2 -19358.43} C_VEL
LIN {X 0,Y 239.546,Z 621.628,A -85,B 0,C 180,E1 -19360.138,E2 -19360.138} C_VEL
LIN {X 0,Y 239.49,Z 622.881,A -85,B 0,C 180,E1 -19361.853,E2 -19361.853} C_VEL
LIN {X 0,Y 239.552,Z 623.957,A -85,B 0,C 180,E1 -19364.498,E2 -19364.498} C_VEL
LIN {X 0,Y 239.688,Z 624.068,A -85,B 0,C 180,E1 -19367.05,E2 -19367.05} C_VEL
LIN {X 0,Y 239.957,Z 623.65,A -85,B 0,C 180,E1 -19368.794,E2 -19368.794} C_VEL
LIN {X 0,Y 240.41,Z 622.662,A -85,B 0,C 180,E1 -19370.696,E2 -19370.696} C_VEL
LIN {X 0,Y 241.569,Z 619.727,A -85,B 0,C 180,E1 -19374.035,E2 -19374.035} C_VEL
LIN {X 0,Y 242.988,Z 616.08,A -85,B 0,C 180,E1 -19376.715,E2 -19376.715} C_VEL
LIN {X 0,Y 244.73,Z 611.486,A -85,B 0,C 180,E1 -19379.221,E2 -19379.221} C_VEL
LIN {X 0,Y 247.01,Z 605.344,A -85,B 0,C 180,E1 -19381.791,E2 -19381.791} C_VEL
LIN {X 0,Y 249.645,Z 597.789,A -85,B 0,C 180,E1 -19384.265,E2 -19384.265} C_VEL
LIN {X 0,Y 252.172,Z 590.124,A -85,B 0,C 180,E1 -19386.264,E2 -19386.264} C_VEL
LIN {X 0,Y 255.211,Z 580.388,A -85,B 0,C 180,E1 -19388.286,E2 -19388.286} C_VEL
LIN {X 0,Y 257.96,Z 570,A -85,B 0,C 180,E1 -19389.988,E2 -19389.988} C_VEL
LIN {X 0,Y 260.409,Z 559.176,A -85,B 0,C 180,E1 -19391.391,E2 -19391.391} C_VEL
LIN {X 0,Y 262.693,Z 546.815,A -85,B 0,C 180,E1 -19392.624,E2 -19392.624} C_VEL
LIN {X 0,Y 264.611,Z 533.714,A -85,B 0,C 180,E1 -19393.541,E2 -19393.541} C_VEL
LIN {X 0,Y 265.98,Z 520.085,A -85,B 0,C 180,E1 -19394.169,E2 -19394.169} C_VEL
LIN {X 0,Y 268.618,Z 461.507,A -85,B 0,C 180,E1 -19395.738,E2 -19395.738} C_VEL
LIN {X 0,Y 263.095,Z 448.806,A -85,B 0,C 180,E1 -19397.119,E2 -19397.119} C_VEL
LIN {X 0,Y 256.329,Z 435.467,A -85,B 0,C 180,E1 -19398.85,E2 -19398.85} C_VEL
LIN {X 0,Y 250.496,Z 425.435,A -85,B 0,C 180,E1 -19400.401,E2 -19400.401} C_VEL
LIN {X 0,Y 245.604,Z 417.54,A -85,B 0,C 180,E1 -19401.775,E2 -19401.775} C_VEL
LIN {X 0,Y 243.39,Z 413.605,A -85,B 0,C 180,E1 -19402.555,E2 -19402.555} C_VEL
LIN {X 0,Y 242.059,Z 409.069,A -85,B 0,C 180,E1 -19405.264,E2 -19405.264} C_VEL
LIN {X 0,Y 241.991,Z 408.84,A -85,B 0,C 180,E1 -19407.374,E2 -19407.374} C_VEL
LIN {X 0,Y 242.009,Z 408.813,A -85,B 0,C 180,E1 -19410.596,E2 -19410.596} C_VEL
LIN {X 0,Y 242.063,Z 408.828,A -85,B 0,C 180,E1 -19414.183,E2 -19414.183} C_VEL
LIN {X 0,Y 242.048,Z 408.826,A -85,B 0,C 180,E1 -19418.297,E2 -19418.297} C_VEL
LIN {X 0,Y 242.158,Z 408.822,A -85,B 0,C 180,E1 -19423.278,E2 -19423.278} C_VEL
LIN {X 0,Y 242.18,Z 408.816,A -85,B 0,C 180,E1 -19428.28,E2 -19428.28} C_VEL
LIN {X 0,Y 242.422,Z 408.788,A -85,B 0,C 180,E1 -19431.666,E2 -19431.666} C_VEL
LIN {X 0,Y 242.263,Z 408.796,A -85,B 0,C 180,E1 -19435.007,E2 -19435.007} C_VEL
LIN {X 0,Y 242.641,Z 408.749,A -85,B 0,C 180,E1 -19438.34,E2 -19438.34} C_VEL
LIN {X 0,Y 242.633,Z 408.762,A -85,B 0,C 180,E1 -19441.66,E2 -19441.66} C_VEL
LIN {X 0,Y 242.427,Z 408.788,A -85,B 0,C 180,E1 -19446.659,E2 -19446.659} C_VEL
LIN {X 0,Y 242.362,Z 408.783,A -85,B 0,C 180,E1 -19449.377,E2 -19449.377} C_VEL
LIN {X 0,Y 241.656,Z 408.882,A -85,B 0,C 180,E1 -19450.762,E2 -19450.762} C_VEL
LIN {X 0,Y 238.698,Z 409.249,A -85,B 0,C 180,E1 -19453.017,E2 -19453.017} C_VEL
LIN {X 0,Y 236.207,Z 409.558,A -85,B 0,C 180,E1 -19454.856,E2 -19454.856} C_VEL
LIN {X 0,Y 235.16,Z 409.694,A -85,B 0,C 180,E1 -19456.285,E2 -19456.285} C_VEL
LIN {X 0,Y 235.086,Z 409.696,A -85,B 0,C 180,E1 -19456.77,E2 -19456.77} C_VEL
LIN {X 0,Y 235.007,Z 409.709,A -85,B 0,C 180,E1 -19461.031,E2 -19461.031} C_VEL
LIN {X 0,Y 234.99,Z 409.704,A -85,B 0,C 180,E1 -19466.207,E2 -19466.207} C_VEL
LIN {X 0,Y 234.928,Z 409.712,A -85,B 0,C 180,E1 -19470.568,E2 -19470.568} C_VEL
LIN {X 0,Y 234.957,Z 409.711,A -85,B 0,C 180,E1 -19474.634,E2 -19474.634} C_VEL
LIN {X 0,Y 234.965,Z 409.718,A -85,B 0,C 180,E1 -19478.953,E2 -19478.953} C_VEL
LIN {X 0,Y 234.964,Z 409.738,A -85,B 0,C 180,E1 -19483.719,E2 -19483.719} C_VEL
LIN {X 0,Y 235.697,Z 412.584,A -85,B 0,C 180,E1 -19485.695,E2 -19485.695} C_VEL
LIN {X 0,Y 237.435,Z 418.434,A -85,B 0,C 180,E1 -19489.096,E2 -19489.096} C_VEL
LIN {X 0,Y 240.196,Z 423.06,A -85,B 0,C 180,E1 -19490.039,E2 -19490.039} C_VEL
LIN {X 0,Y 246.49,Z 433.625,A -85,B 0,C 180,E1 -19491.917,E2 -19491.917} C_VEL
LIN {X 0,Y 254.631,Z 448.998,A -85,B 0,C 180,E1 -19494.172,E2 -19494.172} C_VEL
LIN {X 0,Y 260.946,Z 463.001,A -85,B 0,C 180,E1 -19495.85,E2 -19495.85} C_VEL
LIN {X 0,Y 261.853,Z 466.527,A -85,B 0,C 180,E1 -19496.134,E2 -19496.134} C_VEL
LIN {X 0,Y 262.605,Z 472.096,A -85,B 0,C 180,E1 -19496.459,E2 -19496.459} C_VEL
LIN {X 0,Y 260.014,Z 526.796,A -85,B 0,C 180,E1 -19497.96,E2 -19497.96} C_VEL
LIN {X 0,Y 258.556,Z 540.431,A -85,B 0,C 180,E1 -19498.608,E2 -19498.608} C_VEL
LIN {X 0,Y 256.727,Z 552.403,A -85,B 0,C 180,E1 -19499.46,E2 -19499.46} C_VEL
LIN {X 0,Y 254.227,Z 564.409,A -85,B 0,C 180,E1 -19500.615,E2 -19500.615} C_VEL
LIN {X 0,Y 251.551,Z 575.821,A -85,B 0,C 180,E1 -19502.098,E2 -19502.098} C_VEL
LIN {X 0,Y 248.61,Z 586.138,A -85,B 0,C 180,E1 -19503.788,E2 -19503.788} C_VEL
LIN {X 0,Y 245.918,Z 594.588,A -85,B 0,C 180,E1 -19505.52,E2 -19505.52} C_VEL
LIN {X 0,Y 242.889,Z 603.478,A -85,B 0,C 180,E1 -19507.808,E2 -19507.808} C_VEL
LIN {X 0,Y 240.239,Z 611.149,A -85,B 0,C 180,E1 -19510.342,E2 -19510.342} C_VEL
LIN {X 0,Y 237.807,Z 617.107,A -85,B 0,C 180,E1 -19512.811,E2 -19512.811} C_VEL
LIN {X 0,Y 235.947,Z 621.831,A -85,B 0,C 180,E1 -19515.335,E2 -19515.335} C_VEL
LIN {X 0,Y 234.58,Z 625.464,A -85,B 0,C 180,E1 -19517.895,E2 -19517.895} C_VEL
LIN {X 0,Y 233.875,Z 627.351,A -85,B 0,C 180,E1 -19519.613,E2 -19519.613} C_VEL
LIN {X 0,Y 233.354,Z 628.8,A -85,B 0,C 180,E1 -19521.34,E2 -19521.34} C_VEL
LIN {X 0,Y 232.769,Z 630.485,A -85,B 0,C 180,E1 -19524.804,E2 -19524.804} C_VEL
LIN {X 0,Y 232.656,Z 630.757,A -85,B 0,C 180,E1 -19526.537,E2 -19526.537} C_VEL
LIN {X 0,Y 232.67,Z 630.63,A -85,B 0,C 180,E1 -19528.27,E2 -19528.27} C_VEL
LIN {X 0,Y 232.725,Z 630.08,A -85,B 0,C 180,E1 -19530,E2 -19530} C_VEL
LIN {X 0,Y 232.67,Z 629.138,A -85,B 0,C 180,E1 -19531.731,E2 -19531.731} C_VEL
LIN {X 0,Y 232.679,Z 626.652,A -85,B 0,C 180,E1 -19534.614,E2 -19534.614} C_VEL
LIN {X 0,Y 233.004,Z 622.487,A -85,B 0,C 180,E1 -19537.801,E2 -19537.801} C_VEL
LIN {X 0,Y 233.588,Z 617.832,A -85,B 0,C 180,E1 -19540.4,E2 -19540.4} C_VEL
LIN {X 0,Y 234.642,Z 610.776,A -85,B 0,C 180,E1 -19543.423,E2 -19543.423} C_VEL
LIN {X 0,Y 236.101,Z 603.133,A -85,B 0,C 180,E1 -19545.983,E2 -19545.983} C_VEL
LIN {X 0,Y 237.569,Z 595.291,A -85,B 0,C 180,E1 -19548.097,E2 -19548.097} C_VEL
LIN {X 0,Y 239.113,Z 585.535,A -85,B 0,C 180,E1 -19550.229,E2 -19550.229} C_VEL
LIN {X 0,Y 240.822,Z 574.97,A -85,B 0,C 180,E1 -19552.07,E2 -19552.07} C_VEL
LIN {X 0,Y 242.718,Z 563.001,A -85,B 0,C 180,E1 -19553.688,E2 -19553.688} C_VEL
LIN {X 0,Y 244.386,Z 550.137,A -85,B 0,C 180,E1 -19554.985,E2 -19554.985} C_VEL
LIN {X 0,Y 245.605,Z 537.148,A -85,B 0,C 180,E1 -19555.93,E2 -19555.93} C_VEL
LIN {X 0,Y 246.404,Z 524.305,A -85,B 0,C 180,E1 -19556.523,E2 -19556.523} C_VEL
LIN {X 0,Y 248.148,Z 464.519,A -85,B 0,C 180,E1 -19558.237,E2 -19558.237} C_VEL
LIN {X 0,Y 244.821,Z 440.092,A -85,B 0,C 180,E1 -19559.348,E2 -19559.348} C_VEL
LIN {X 0,Y 239.006,Z 424.215,A -85,B 0,C 180,E1 -19560.498,E2 -19560.498} C_VEL
LIN {X 0,Y 236.972,Z 419.024,A -85,B 0,C 180,E1 -19560.969,E2 -19560.969} C_VEL
LIN {X 0,Y 235.736,Z 413.038,A -85,B 0,C 180,E1 -19563.408,E2 -19563.408} C_VEL
LIN {X 0,Y 235.004,Z 409.74,A -85,B 0,C 180,E1 -19564.976,E2 -19564.976} C_VEL
LIN {X 0,Y 234.942,Z 409.703,A -85,B 0,C 180,E1 -19568.944,E2 -19568.944} C_VEL
LIN {X 0,Y 234.958,Z 409.705,A -85,B 0,C 180,E1 -19573.469,E2 -19573.469} C_VEL
LIN {X 0,Y 234.964,Z 409.679,A -85,B 0,C 180,E1 -19576.532,E2 -19576.532} C_VEL
LIN {X 0,Y 234.955,Z 409.719,A -85,B 0,C 180,E1 -19581.086,E2 -19581.086} C_VEL
LIN {X 0,Y 234.96,Z 409.71,A -85,B 0,C 180,E1 -19585.367,E2 -19585.367} C_VEL
LIN {X 0,Y 234.922,Z 409.716,A -85,B 0,C 180,E1 -19589.431,E2 -19589.431} C_VEL
LIN {X 0,Y 234.992,Z 409.712,A -85,B 0,C 180,E1 -19593.794,E2 -19593.794} C_VEL
LIN {X 0,Y 234.996,Z 409.695,A -85,B 0,C 180,E1 -19598.968,E2 -19598.968} C_VEL
LIN {X 0,Y 235.094,Z 409.697,A -85,B 0,C 180,E1 -19603.059,E2 -19603.059} C_VEL
LIN {X 0,Y 235.111,Z 409.683,A -85,B 0,C 180,E1 -19607.922,E2 -19607.922} C_VEL
LIN {X 0,Y 235.329,Z 409.654,A -85,B 0,C 180,E1 -19611.412,E2 -19611.412} C_VEL
LIN {X 0,Y 235.371,Z 409.66,A -85,B 0,C 180,E1 -19613.14,E2 -19613.14} C_VEL
LIN {X 0,Y 235.593,Z 409.628,A -85,B 0,C 180,E1 -19618.29,E2 -19618.29} C_VEL
LIN {X 0,Y 235.593,Z 409.613,A -85,B 0,C 180,E1 -19621.709,E2 -19621.709} C_VEL
LIN {X 0,Y 235.39,Z 409.663,A -85,B 0,C 180,E1 -19626.859,E2 -19626.859} C_VEL
LIN {X 0,Y 235.212,Z 409.673,A -85,B 0,C 180,E1 -19630.328,E2 -19630.328} C_VEL
LIN {X 0,Y 235.109,Z 409.691,A -85,B 0,C 180,E1 -19635.607,E2 -19635.607} C_VEL
LIN {X 0,Y 235.006,Z 409.71,A -85,B 0,C 180,E1 -19639.206,E2 -19639.206} C_VEL
LIN {X 0,Y 234.959,Z 409.694,A -85,B 0,C 180,E1 -19642.883,E2 -19642.883} C_VEL
LIN {X 0,Y 234.968,Z 409.708,A -85,B 0,C 180,E1 -19646.657,E2 -19646.657} C_VEL
LIN {X 0,Y 234.93,Z 409.718,A -85,B 0,C 180,E1 -19650.568,E2 -19650.568} C_VEL
LIN {X 0,Y 234.928,Z 409.703,A -85,B 0,C 180,E1 -19654.638,E2 -19654.638} C_VEL
LIN {X 0,Y 234.941,Z 409.72,A -85,B 0,C 180,E1 -19658.945,E2 -19658.945} C_VEL
LIN {X 0,Y 234.889,Z 409.716,A -85,B 0,C 180,E1 -19663.485,E2 -19663.485} C_VEL
LIN {X 0,Y 234.945,Z 409.72,A -85,B 0,C 180,E1 -19666.528,E2 -19666.528} C_VEL
LIN {X 0,Y 234.955,Z 409.717,A -85,B 0,C 180,E1 -19671.086,E2 -19671.086} C_VEL
LIN {X 0,Y 234.961,Z 409.697,A -85,B 0,C 180,E1 -19675.367,E2 -19675.367} C_VEL
LIN {X 0,Y 234.97,Z 409.708,A -85,B 0,C 180,E1 -19680.157,E2 -19680.157} C_VEL
LIN {X 0,Y 234.995,Z 409.695,A -85,B 0,C 180,E1 -19683.794,E2 -19683.794} C_VEL
LIN {X 0,Y 235.012,Z 409.703,A -85,B 0,C 180,E1 -19688.97,E2 -19688.97} C_VEL
LIN {X 0,Y 235.07,Z 409.815,A -85,B 0,C 180,E1 -19690.459,E2 -19690.459} C_VEL
LIN {X 0,Y 235.852,Z 413.34,A -85,B 0,C 180,E1 -19691.968,E2 -19691.968} C_VEL
LIN {X 0,Y 242.016,Z 428.57,A -85,B 0,C 180,E1 -19693.233,E2 -19693.233} C_VEL
LIN {X 0,Y 246.671,Z 442.274,A -85,B 0,C 180,E1 -19694.17,E2 -19694.17} C_VEL
LIN {X 0,Y 248.503,Z 454.127,A -85,B 0,C 180,E1 -19694.729,E2 -19694.729} C_VEL
LIN {X 0,Y 246.333,Z 520.58,A -85,B 0,C 180,E1 -19696.635,E2 -19696.635} C_VEL
LIN {X 0,Y 245.471,Z 533.56,A -85,B 0,C 180,E1 -19697.316,E2 -19697.316} C_VEL
LIN {X 0,Y 244.3,Z 545.466,A -85,B 0,C 180,E1 -19698.235,E2 -19698.235} C_VEL
LIN {X 0,Y 242.745,Z 557.79,A -85,B 0,C 180,E1 -19699.532,E2 -19699.532} C_VEL
LIN {X 0,Y 241.046,Z 568.39,A -85,B 0,C 180,E1 -19700.983,E2 -19700.983} C_VEL
LIN {X 0,Y 239.469,Z 577.934,A -85,B 0,C 180,E1 -19702.623,E2 -19702.623} C_VEL
LIN {X 0,Y 237.928,Z 586.785,A -85,B 0,C 180,E1 -19704.491,E2 -19704.491} C_VEL
LIN {X 0,Y 236.52,Z 594.914,A -85,B 0,C 180,E1 -19706.593,E2 -19706.593} C_VEL
LIN {X 0,Y 235.011,Z 602.914,A -85,B 0,C 180,E1 -19709.143,E2 -19709.143} C_VEL
LIN {X 0,Y 234.004,Z 609.291,A -85,B 0,C 180,E1 -19711.721,E2 -19711.721} C_VEL
LIN {X 0,Y 233.329,Z 614.361,A -85,B 0,C 180,E1 -19714.318,E2 -19714.318} C_VEL
LIN {X 0,Y 232.861,Z 618.299,A -85,B 0,C 180,E1 -19716.933,E2 -19716.933} C_VEL
LIN {X 0,Y 232.571,Z 620.334,A -85,B 0,C 180,E1 -19718.69,E2 -19718.69} C_VEL
LIN {X 0,Y 232.42,Z 621.947,A -85,B 0,C 180,E1 -19720.452,E2 -19720.452} C_VEL
LIN {X 0,Y 232.401,Z 623.13,A -85,B 0,C 180,E1 -19722.22,E2 -19722.22} C_VEL
LIN {X 0,Y 232.458,Z 624.05,A -85,B 0,C 180,E1 -19724.654,E2 -19724.654} C_VEL
LIN {X 0,Y 232.659,Z 624.147,A -85,B 0,C 180,E1 -19727.581,E2 -19727.581} C_VEL
LIN {X 0,Y 232.99,Z 623.638,A -85,B 0,C 180,E1 -19729.378,E2 -19729.378} C_VEL
LIN {X 0,Y 233.433,Z 622.698,A -85,B 0,C 180,E1 -19731.178,E2 -19731.178} C_VEL
LIN {X 0,Y 234.02,Z 621.342,A -85,B 0,C 180,E1 -19732.979,E2 -19732.979} C_VEL
LIN {X 0,Y 235.26,Z 618.432,A -85,B 0,C 180,E1 -19735.667,E2 -19735.667} C_VEL
LIN {X 0,Y 236.893,Z 614.413,A -85,B 0,C 180,E1 -19738.337,E2 -19738.337} C_VEL
LIN {X 0,Y 239.025,Z 609.202,A -85,B 0,C 180,E1 -19740.949,E2 -19740.949} C_VEL
LIN {X 0,Y 241.535,Z 602.457,A -85,B 0,C 180,E1 -19743.561,E2 -19743.561} C_VEL
LIN {X 0,Y 244.483,Z 594.38,A -85,B 0,C 180,E1 -19745.996,E2 -19745.996} C_VEL
LIN {X 0,Y 247.513,Z 585.389,A -85,B 0,C 180,E1 -19748.138,E2 -19748.138} C_VEL
LIN {X 0,Y 250.37,Z 575.815,A -85,B 0,C 180,E1 -19749.948,E2 -19749.948} C_VEL
LIN {X 0,Y 253.221,Z 564.993,A -85,B 0,C 180,E1 -19751.555,E2 -19751.555} C_VEL
LIN {X 0,Y 255.625,Z 553.71,A -85,B 0,C 180,E1 -19752.878,E2 -19752.878} C_VEL
LIN {X 0,Y 257.741,Z 541.894,A -85,B 0,C 180,E1 -19753.916,E2 -19753.916} C_VEL
LIN {X 0,Y 259.441,Z 529.097,A -85,B 0,C 180,E1 -19754.704,E2 -19754.704} C_VEL
LIN {X 0,Y 260.556,Z 516.03,A -85,B 0,C 180,E1 -19755.212,E2 -19755.212} C_VEL
LIN {X 0,Y 262.871,Z 463.422,A -85,B 0,C 180,E1 -19756.647,E2 -19756.647} C_VEL
LIN {X 0,Y 256.69,Z 449.471,A -85,B 0,C 180,E1 -19758.267,E2 -19758.267} C_VEL
LIN {X 0,Y 249.567,Z 435.86,A -85,B 0,C 180,E1 -19760.192,E2 -19760.192} C_VEL
LIN {X 0,Y 242.087,Z 423.171,A -85,B 0,C 180,E1 -19762.358,E2 -19762.358} C_VEL
LIN {X 0,Y 238.469,Z 417.74,A -85,B 0,C 180,E1 -19763.463,E2 -19763.463} C_VEL
LIN {X 0,Y 236.231,Z 413.88,A -85,B 0,C 180,E1 -19764.281,E2 -19764.281} C_VEL
LIN {X 0,Y 234.96,Z 409.778,A -85,B 0,C 180,E1 -19766.945,E2 -19766.945} C_VEL
LIN {X 0,Y 234.932,Z 409.699,A -85,B 0,C 180,E1 -19771.403,E2 -19771.403} C_VEL
LIN {X 0,Y 234.982,Z 409.71,A -85,B 0,C 180,E1 -19775.246,E2 -19775.246} C_VEL
LIN {X 0,Y 235.007,Z 409.707,A -85,B 0,C 180,E1 -19778.97,E2 -19778.97} C_VEL
LIN {X 0,Y 235.091,Z 409.699,A -85,B 0,C 180,E1 -19783.059,E2 -19783.059} C_VEL
LIN {X 0,Y 235.14,Z 409.695,A -85,B 0,C 180,E1 -19787.923,E2 -19787.923} C_VEL
LIN {X 0,Y 235.371,Z 409.664,A -85,B 0,C 180,E1 -19791.414,E2 -19791.414} C_VEL
LIN {X 0,Y 235.399,Z 409.656,A -85,B 0,C 180,E1 -19793.141,E2 -19793.141} C_VEL
LIN {X 0,Y 235.601,Z 409.626,A -85,B 0,C 180,E1 -19798.291,E2 -19798.291} C_VEL
LIN {X 0,Y 235.593,Z 409.639,A -85,B 0,C 180,E1 -19801.71,E2 -19801.71} C_VEL
LIN {X 0,Y 235.398,Z 409.661,A -85,B 0,C 180,E1 -19806.859,E2 -19806.859} C_VEL
LIN {X 0,Y 235.233,Z 409.679,A -85,B 0,C 180,E1 -19810.327,E2 -19810.327} C_VEL
LIN {X 0,Y 235.108,Z 409.699,A -85,B 0,C 180,E1 -19815.607,E2 -19815.607} C_VEL
LIN {X 0,Y 235.086,Z 409.696,A -85,B 0,C 180,E1 -19816.77,E2 -19816.77} C_VEL
LIN {X 0,Y 234.432,Z 409.78,A -85,B 0,C 180,E1 -19818.201,E2 -19818.201} C_VEL
LIN {X 0,Y 231.526,Z 410.146,A -85,B 0,C 180,E1 -19820.531,E2 -19820.531} C_VEL
LIN {X 0,Y 229.039,Z 410.449,A -85,B 0,C 180,E1 -19822.433,E2 -19822.433} C_VEL
LIN {X 0,Y 227.97,Z 410.581,A -85,B 0,C 180,E1 -19823.91,E2 -19823.91} C_VEL
LIN {X 0,Y 227.884,Z 410.588,A -85,B 0,C 180,E1 -19824.412,E2 -19824.412} C_VEL
LIN {X 0,Y 227.882,Z 410.59,A -85,B 0,C 180,E1 -19827.556,E2 -19827.556} C_VEL
LIN {X 0,Y 227.869,Z 410.595,A -85,B 0,C 180,E1 -19831.623,E2 -19831.623} C_VEL
LIN {X 0,Y 227.899,Z 410.599,A -85,B 0,C 180,E1 -19835.869,E2 -19835.869} C_VEL
LIN {X 0,Y 227.892,Z 410.577,A -85,B 0,C 180,E1 -19840.363,E2 -19840.363} C_VEL
LIN {X 0,Y 227.939,Z 410.752,A -85,B 0,C 180,E1 -19842.272,E2 -19842.272} C_VEL
LIN {X 0,Y 229.91,Z 417.673,A -85,B 0,C 180,E1 -19846.871,E2 -19846.871} C_VEL
LIN {X 0,Y 230.431,Z 418.967,A -85,B 0,C 180,E1 -19847.316,E2 -19847.316} C_VEL
LIN {X 0,Y 233.293,Z 423.336,A -85,B 0,C 180,E1 -19848.31,E2 -19848.31} C_VEL
LIN {X 0,Y 240.022,Z 434.429,A -85,B 0,C 180,E1 -19850.477,E2 -19850.477} C_VEL
LIN {X 0,Y 245.35,Z 444.204,A -85,B 0,C 180,E1 -19852.088,E2 -19852.088} C_VEL
LIN {X 0,Y 251.047,Z 455.527,A -85,B 0,C 180,E1 -19853.712,E2 -19853.712} C_VEL
LIN {X 0,Y 256.014,Z 466.752,A -85,B 0,C 180,E1 -19855.086,E2 -19855.086} C_VEL
LIN {X 0,Y 257.044,Z 473.01,A -85,B 0,C 180,E1 -19855.503,E2 -19855.503} C_VEL
LIN {X 0,Y 254.405,Z 526.546,A -85,B 0,C 180,E1 -19856.994,E2 -19856.994} C_VEL
LIN {X 0,Y 252.913,Z 540.133,A -85,B 0,C 180,E1 -19857.646,E2 -19857.646} C_VEL
LIN {X 0,Y 250.903,Z 552.733,A -85,B 0,C 180,E1 -19858.555,E2 -19858.555} C_VEL
LIN {X 0,Y 248.504,Z 563.825,A -85,B 0,C 180,E1 -19859.635,E2 -19859.635} C_VEL
LIN {X 0,Y 245.665,Z 575.331,A -85,B 0,C 180,E1 -19861.135,E2 -19861.135} C_VEL
LIN {X 0,Y 242.633,Z 585.711,A -85,B 0,C 180,E1 -19862.858,E2 -19862.858} C_VEL
LIN {X 0,Y 239.49,Z 595.092,A -85,B 0,C 180,E1 -19864.818,E2 -19864.818} C_VEL
LIN {X 0,Y 236.234,Z 604.136,A -85,B 0,C 180,E1 -19867.248,E2 -19867.248} C_VEL
LIN {X 0,Y 233.558,Z 611.435,A -85,B 0,C 180,E1 -19869.755,E2 -19869.755} C_VEL
LIN {X 0,Y 231.027,Z 617.32,A -85,B 0,C 180,E1 -19872.29,E2 -19872.29} C_VEL
LIN {X 0,Y 229.063,Z 621.977,A -85,B 0,C 180,E1 -19874.884,E2 -19874.884} C_VEL
LIN {X 0,Y 227.619,Z 625.547,A -85,B 0,C 180,E1 -19877.519,E2 -19877.519} C_VEL
LIN {X 0,Y 226.878,Z 627.399,A -85,B 0,C 180,E1 -19879.289,E2 -19879.289} C_VEL
LIN {X 0,Y 225.937,Z 629.801,A -85,B 0,C 180,E1 -19882.853,E2 -19882.853} C_VEL
LIN {X 0,Y 225.572,Z 630.668,A -85,B 0,C 180,E1 -19886.428,E2 -19886.428} C_VEL
LIN {X 0,Y 225.57,Z 630.489,A -85,B 0,C 180,E1 -19888.215,E2 -19888.215} C_VEL
LIN {X 0,Y 225.641,Z 629.912,A -85,B 0,C 180,E1 -19890,E2 -19890} C_VEL
LIN {X 0,Y 225.57,Z 628.943,A -85,B 0,C 180,E1 -19891.786,E2 -19891.786} C_VEL
LIN {X 0,Y 225.57,Z 626.736,A -85,B 0,C 180,E1 -19894.427,E2 -19894.427} C_VEL
LIN {X 0,Y 225.821,Z 623.451,A -85,B 0,C 180,E1 -19897.151,E2 -19897.151} C_VEL
LIN {X 0,Y 226.338,Z 619.121,A -85,B 0,C 180,E1 -19899.833,E2 -19899.833} C_VEL
LIN {X 0,Y 227.168,Z 613.579,A -85,B 0,C 180,E1 -19902.507,E2 -19902.507} C_VEL
LIN {X 0,Y 228.431,Z 606.642,A -85,B 0,C 180,E1 -19905.16,E2 -19905.16} C_VEL
LIN {X 0,Y 229.737,Z 599.536,A -85,B 0,C 180,E1 -19907.354,E2 -19907.354} C_VEL
LIN {X 0,Y 231.346,Z 590.942,A -85,B 0,C 180,E1 -19909.522,E2 -19909.522} C_VEL
LIN {X 0,Y 233.172,Z 580.287,A -85,B 0,C 180,E1 -19911.668,E2 -19911.668} C_VEL
LIN {X 0,Y 234.937,Z 569.725,A -85,B 0,C 180,E1 -19913.351,E2 -19913.351} C_VEL
LIN {X 0,Y 236.697,Z 558.063,A -85,B 0,C 180,E1 -19914.797,E2 -19914.797} C_VEL
LIN {X 0,Y 238.149,Z 545.907,A -85,B 0,C 180,E1 -19915.921,E2 -19915.921} C_VEL
LIN {X 0,Y 239.25,Z 533.604,A -85,B 0,C 180,E1 -19916.731,E2 -19916.731} C_VEL
LIN {X 0,Y 239.97,Z 521.569,A -85,B 0,C 180,E1 -19917.233,E2 -19917.233} C_VEL
LIN {X 0,Y 241.618,Z 465.295,A -85,B 0,C 180,E1 -19918.878,E2 -19918.878} C_VEL
LIN {X 0,Y 238.47,Z 442.097,A -85,B 0,C 180,E1 -19919.974,E2 -19919.974} C_VEL
LIN {X 0,Y 232.444,Z 425.654,A -85,B 0,C 180,E1 -19921.22,E2 -19921.22} C_VEL
LIN {X 0,Y 229.762,Z 419.037,A -85,B 0,C 180,E1 -19921.829,E2 -19921.829} C_VEL
LIN {X 0,Y 229.19,Z 416.283,A -85,B 0,C 180,E1 -19922.894,E2 -19922.894} C_VEL
LIN {X 0,Y 227.942,Z 410.622,A -85,B 0,C 180,E1 -19925.563,E2 -19925.563} C_VEL
LIN {X 0,Y 227.843,Z 410.596,A -85,B 0,C 180,E1 -19930.373,E2 -19930.373} C_VEL
LIN {X 0,Y 227.9,Z 410.592,A -85,B 0,C 180,E1 -19932.721,E2 -19932.721} C_VEL
LIN {X 0,Y 227.909,Z 410.567,A -85,B 0,C 180,E1 -19937.738,E2 -19937.738} C_VEL
LIN {X 0,Y 227.871,Z 410.599,A -85,B 0,C 180,E1 -19941.914,E2 -19941.914} C_VEL
LIN {X 0,Y 227.89,Z 410.598,A -85,B 0,C 180,E1 -19946.372,E2 -19946.372} C_VEL
LIN {X 0,Y 227.903,Z 410.584,A -85,B 0,C 180,E1 -19950.435,E2 -19950.435} C_VEL
LIN {X 0,Y 227.923,Z 410.593,A -85,B 0,C 180,E1 -19954.425,E2 -19954.425} C_VEL
LIN {X 0,Y 227.946,Z 410.578,A -85,B 0,C 180,E1 -19958.285,E2 -19958.285} C_VEL
LIN {X 0,Y 228.033,Z 410.575,A -85,B 0,C 180,E1 -19962.826,E2 -19962.826} C_VEL
LIN {X 0,Y 228.069,Z 410.562,A -85,B 0,C 180,E1 -19967.543,E2 -19967.543} C_VEL
LIN {X 0,Y 228.265,Z 410.531,A -85,B 0,C 180,E1 -19971.144,E2 -19971.144} C_VEL
LIN {X 0,Y 228.321,Z 410.537,A -85,B 0,C 180,E1 -19972.927,E2 -19972.927} C_VEL
LIN {X 0,Y 228.552,Z 410.505,A -85,B 0,C 180,E1 -19978.238,E2 -19978.238} C_VEL
LIN {X 0,Y 228.552,Z 410.489,A -85,B 0,C 180,E1 -19981.762,E2 -19981.762} C_VEL
LIN {X 0,Y 228.337,Z 410.543,A -85,B 0,C 180,E1 -19987.072,E2 -19987.072} C_VEL
LIN {X 0,Y 228.143,Z 410.547,A -85,B 0,C 180,E1 -19990.651,E2 -19990.651} C_VEL
LIN {X 0,Y 228.06,Z 410.559,A -85,B 0,C 180,E1 -19994.272,E2 -19994.272} C_VEL
LIN {X 0,Y 228.001,Z 410.583,A -85,B 0,C 180,E1 -19997.953,E2 -19997.953} C_VEL
LIN {X 0,Y 227.928,Z 410.573,A -85,B 0,C 180,E1 -20002.329,E2 -20002.329} C_VEL
LIN {X 0,Y 227.941,Z 410.582,A -85,B 0,C 180,E1 -20006.603,E2 -20006.603} C_VEL
LIN {X 0,Y 227.907,Z 410.592,A -85,B 0,C 180,E1 -20010.296,E2 -20010.296} C_VEL
LIN {X 0,Y 227.876,Z 410.577,A -85,B 0,C 180,E1 -20013.721,E2 -20013.721} C_VEL
LIN {X 0,Y 227.843,Z 410.603,A -85,B 0,C 180,E1 -20018.091,E2 -20018.091} C_VEL
LIN {X 0,Y 227.811,Z 410.59,A -85,B 0,C 180,E1 -20022.742,E2 -20022.742} C_VEL
LIN {X 0,Y 227.892,Z 410.593,A -85,B 0,C 180,E1 -20027.277,E2 -20027.277} C_VEL
LIN {X 0,Y 227.871,Z 410.602,A -85,B 0,C 180,E1 -20031.915,E2 -20031.915} C_VEL
LIN {X 0,Y 227.89,Z 410.562,A -85,B 0,C 180,E1 -20036.373,E2 -20036.373} C_VEL
LIN {X 0,Y 227.92,Z 410.589,A -85,B 0,C 180,E1 -20040.438,E2 -20040.438} C_VEL
LIN {X 0,Y 227.929,Z 410.568,A -85,B 0,C 180,E1 -20044.426,E2 -20044.426} C_VEL
LIN {X 0,Y 227.994,Z 410.6,A -85,B 0,C 180,E1 -20049.709,E2 -20049.709} C_VEL
LIN {X 0,Y 228.137,Z 411.281,A -85,B 0,C 180,E1 -20050.192,E2 -20050.192} C_VEL
LIN {X 0,Y 228.683,Z 413.461,A -85,B 0,C 180,E1 -20051.087,E2 -20051.087} C_VEL
LIN {X 0,Y 235.702,Z 430.605,A -85,B 0,C 180,E1 -20052.583,E2 -20052.583} C_VEL
LIN {X 0,Y 240.332,Z 444.161,A -85,B 0,C 180,E1 -20053.555,E2 -20053.555} C_VEL
LIN {X 0,Y 242.016,Z 456.537,A -85,B 0,C 180,E1 -20054.137,E2 -20054.137} C_VEL
LIN {X 0,Y 239.777,Z 520.481,A -85,B 0,C 180,E1 -20056.007,E2 -20056.007} C_VEL
LIN {X 0,Y 238.852,Z 533.477,A -85,B 0,C 180,E1 -20056.698,E2 -20056.698} C_VEL
LIN {X 0,Y 237.644,Z 545.485,A -85,B 0,C 180,E1 -20057.645,E2 -20057.645} C_VEL
LIN {X 0,Y 236.023,Z 557.96,A -85,B 0,C 180,E1 -20058.992,E2 -20058.992} C_VEL
LIN {X 0,Y 234.249,Z 568.678,A -85,B 0,C 180,E1 -20060.502,E2 -20060.502} C_VEL
LIN {X 0,Y 232.616,Z 578.192,A -85,B 0,C 180,E1 -20062.186,E2 -20062.186} C_VEL
LIN {X 0,Y 230.831,Z 587.917,A -85,B 0,C 180,E1 -20064.321,E2 -20064.321} C_VEL
LIN {X 0,Y 229.433,Z 595.872,A -85,B 0,C 180,E1 -20066.487,E2 -20066.487} C_VEL
LIN {X 0,Y 227.886,Z 603.683,A -85,B 0,C 180,E1 -20069.116,E2 -20069.116} C_VEL
LIN {X 0,Y 226.851,Z 609.921,A -85,B 0,C 180,E1 -20071.775,E2 -20071.775} C_VEL
LIN {X 0,Y 226.213,Z 614.877,A -85,B 0,C 180,E1 -20074.454,E2 -20074.454} C_VEL
LIN {X 0,Y 225.719,Z 618.714,A -85,B 0,C 180,E1 -20077.154,E2 -20077.154} C_VEL
LIN {X 0,Y 225.436,Z 620.699,A -85,B 0,C 180,E1 -20078.967,E2 -20078.967} C_VEL
LIN {X 0,Y 225.3,Z 622.259,A -85,B 0,C 180,E1 -20080.787,E2 -20080.787} C_VEL
LIN {X 0,Y 225.305,Z 623.351,A -85,B 0,C 180,E1 -20082.612,E2 -20082.612} C_VEL
LIN {X 0,Y 225.358,Z 624.139,A -85,B 0,C 180,E1 -20084.814,E2 -20084.814} C_VEL
LIN {X 0,Y 225.637,Z 624.203,A -85,B 0,C 180,E1 -20088.147,E2 -20088.147} C_VEL
LIN {X 0,Y 226.376,Z 622.947,A -85,B 0,C 180,E1 -20091.351,E2 -20091.351} C_VEL
LIN {X 0,Y 227.19,Z 621.224,A -85,B 0,C 180,E1 -20093.712,E2 -20093.712} C_VEL
LIN {X 0,Y 228.964,Z 617.336,A -85,B 0,C 180,E1 -20097.108,E2 -20097.108} C_VEL
LIN {X 0,Y 231.088,Z 612.408,A -85,B 0,C 180,E1 -20100.119,E2 -20100.119} C_VEL
LIN {X 0,Y 233.52,Z 606.582,A -85,B 0,C 180,E1 -20102.8,E2 -20102.8} C_VEL
LIN {X 0,Y 236.431,Z 599.183,A -85,B 0,C 180,E1 -20105.424,E2 -20105.424} C_VEL
LIN {X 0,Y 239.454,Z 590.944,A -85,B 0,C 180,E1 -20107.72,E2 -20107.72} C_VEL
LIN {X 0,Y 242.741,Z 581.328,A -85,B 0,C 180,E1 -20109.833,E2 -20109.833} C_VEL
LIN {X 0,Y 245.57,Z 571.69,A -85,B 0,C 180,E1 -20111.518,E2 -20111.518} C_VEL
LIN {X 0,Y 248.389,Z 560.549,A -85,B 0,C 180,E1 -20113.045,E2 -20113.045} C_VEL
LIN {X 0,Y 250.823,Z 548.524,A -85,B 0,C 180,E1 -20114.325,E2 -20114.325} C_VEL
LIN {X 0,Y 252.899,Z 536.199,A -85,B 0,C 180,E1 -20115.264,E2 -20115.264} C_VEL
LIN {X 0,Y 254.411,Z 522.656,A -85,B 0,C 180,E1 -20115.96,E2 -20115.96} C_VEL
LIN {X 0,Y 255.73,Z 499.569,A -85,B 0,C 180,E1 -20116.633,E2 -20116.633} C_VEL
LIN {X 0,Y 257.293,Z 465.507,A -85,B 0,C 180,E1 -20117.573,E2 -20117.573} C_VEL
LIN {X 0,Y 250.497,Z 450.554,A -85,B 0,C 180,E1 -20119.438,E2 -20119.438} C_VEL
LIN {X 0,Y 243.921,Z 438.139,A -85,B 0,C 180,E1 -20121.322,E2 -20121.322} C_VEL
LIN {X 0,Y 237.822,Z 427.797,A -85,B 0,C 180,E1 -20123.19,E2 -20123.19} C_VEL
LIN {X 0,Y 234.723,Z 422.991,A -85,B 0,C 180,E1 -20124.184,E2 -20124.184} C_VEL
LIN {X 0,Y 231.54,Z 418.214,A -85,B 0,C 180,E1 -20125.245,E2 -20125.245} C_VEL
LIN {X 0,Y 228.846,Z 413.98,A -85,B 0,C 180,E1 -20126.298,E2 -20126.298} C_VEL
LIN {X 0,Y 227.894,Z 410.678,A -85,B 0,C 180,E1 -20128.57,E2 -20128.57} C_VEL
LIN {X 0,Y 227.937,Z 410.593,A -85,B 0,C 180,E1 -20133.397,E2 -20133.397} C_VEL
LIN {X 0,Y 227.957,Z 410.581,A -85,B 0,C 180,E1 -20138.287,E2 -20138.287} C_VEL
LIN {X 0,Y 228.029,Z 410.577,A -85,B 0,C 180,E1 -20142.826,E2 -20142.826} C_VEL
LIN {X 0,Y 228.087,Z 410.574,A -85,B 0,C 180,E1 -20147.544,E2 -20147.544} C_VEL
LIN {X 0,Y 228.3,Z 410.541,A -85,B 0,C 180,E1 -20151.146,E2 -20151.146} C_VEL
LIN {X 0,Y 228.35,Z 410.536,A -85,B 0,C 180,E1 -20152.929,E2 -20152.929} C_VEL
LIN {X 0,Y 228.56,Z 410.503,A -85,B 0,C 180,E1 -20158.238,E2 -20158.238} C_VEL
LIN {X 0,Y 228.551,Z 410.516,A -85,B 0,C 180,E1 -20161.762,E2 -20161.762} C_VEL
LIN {X 0,Y 228.349,Z 410.538,A -85,B 0,C 180,E1 -20167.072,E2 -20167.072} C_VEL
LIN {X 0,Y 228.158,Z 410.562,A -85,B 0,C 180,E1 -20170.651,E2 -20170.651} C_VEL
LIN {X 0,Y 228.059,Z 410.563,A -85,B 0,C 180,E1 -20174.273,E2 -20174.273} C_VEL
LIN {X 0,Y 227.998,Z 410.571,A -85,B 0,C 180,E1 -20177.954,E2 -20177.954} C_VEL
LIN {X 0,Y 227.925,Z 410.581,A -85,B 0,C 180,E1 -20182.33,E2 -20182.33} C_VEL
LIN {X 0,Y 227.884,Z 410.588,A -85,B 0,C 180,E1 -20184.412,E2 -20184.412} C_VEL
LIN {X 0,Y 227.21,Z 410.679,A -85,B 0,C 180,E1 -20185.886,E2 -20185.886} C_VEL
LIN {X 0,Y 224.337,Z 411.039,A -85,B 0,C 180,E1 -20188.291,E2 -20188.291} C_VEL
LIN {X 0,Y 221.906,Z 411.334,A -85,B 0,C 180,E1 -20190.253,E2 -20190.253} C_VEL
LIN {X 0,Y 220.881,Z 411.467,A -85,B 0,C 180,E1 -20191.777,E2 -20191.777} C_VEL
LIN {X 0,Y 220.806,Z 411.475,A -85,B 0,C 180,E1 -20192.294,E2 -20192.294} C_VEL
LIN {X 0,Y 220.865,Z 411.466,A -85,B 0,C 180,E1 -20197.299,E2 -20197.299} C_VEL
LIN {X 0,Y 220.894,Z 411.699,A -85,B 0,C 180,E1 -20200.511,E2 -20200.511} C_VEL
LIN {X 0,Y 222.702,Z 417.832,A -85,B 0,C 180,E1 -20204.878,E2 -20204.878} C_VEL
LIN {X 0,Y 224.758,Z 421.578,A -85,B 0,C 180,E1 -20205.831,E2 -20205.831} C_VEL
LIN {X 0,Y 226.942,Z 424.601,A -85,B 0,C 180,E1 -20206.618,E2 -20206.618} C_VEL
LIN {X 0,Y 230.786,Z 430.704,A -85,B 0,C 180,E1 -20207.975,E2 -20207.975} C_VEL
LIN {X 0,Y 235.749,Z 438.872,A -85,B 0,C 180,E1 -20209.626,E2 -20209.626} C_VEL
LIN {X 0,Y 241.339,Z 449.34,A -85,B 0,C 180,E1 -20211.401,E2 -20211.401} C_VEL
LIN {X 0,Y 246.963,Z 460.806,A -85,B 0,C 180,E1 -20213.081,E2 -20213.081} C_VEL
LIN {X 0,Y 251.054,Z 470.443,A -85,B 0,C 180,E1 -20214.275,E2 -20214.275} C_VEL
LIN {X 0,Y 251.536,Z 474.325,A -85,B 0,C 180,E1 -20214.514,E2 -20214.514} C_VEL
LIN {X 0,Y 248.866,Z 526.269,A -85,B 0,C 180,E1 -20215.976,E2 -20215.976} C_VEL
LIN {X 0,Y 247.351,Z 539.718,A -85,B 0,C 180,E1 -20216.625,E2 -20216.625} C_VEL
LIN {X 0,Y 245.366,Z 552,A -85,B 0,C 180,E1 -20217.518,E2 -20217.518} C_VEL
LIN {X 0,Y 242.86,Z 563.271,A -85,B 0,C 180,E1 -20218.609,E2 -20218.609} C_VEL
LIN {X 0,Y 240.296,Z 573.58,A -85,B 0,C 180,E1 -20219.944,E2 -20219.944} C_VEL
LIN {X 0,Y 237.075,Z 584.242,A -85,B 0,C 180,E1 -20221.686,E2 -20221.686} C_VEL
LIN {X 0,Y 233.771,Z 593.855,A -85,B 0,C 180,E1 -20223.678,E2 -20223.678} C_VEL
LIN {X 0,Y 230.794,Z 601.75,A -85,B 0,C 180,E1 -20225.727,E2 -20225.727} C_VEL
LIN {X 0,Y 227.742,Z 609.505,A -85,B 0,C 180,E1 -20228.266,E2 -20228.266} C_VEL
LIN {X 0,Y 225.105,Z 615.73,A -85,B 0,C 180,E1 -20230.864,E2 -20230.864} C_VEL
LIN {X 0,Y 222.808,Z 620.704,A -85,B 0,C 180,E1 -20233.509,E2 -20233.509} C_VEL
LIN {X 0,Y 221.165,Z 624.568,A -85,B 0,C 180,E1 -20236.213,E2 -20236.213} C_VEL
LIN {X 0,Y 219.898,Z 627.431,A -85,B 0,C 180,E1 -20238.945,E2 -20238.945} C_VEL
LIN {X 0,Y 218.872,Z 629.77,A -85,B 0,C 180,E1 -20242.621,E2 -20242.621} C_VEL
LIN {X 0,Y 218.542,Z 630.508,A -85,B 0,C 180,E1 -20245.504,E2 -20245.504} C_VEL
LIN {X 0,Y 218.473,Z 630.346,A -85,B 0,C 180,E1 -20248.157,E2 -20248.157} C_VEL
LIN {X 0,Y 218.558,Z 629.743,A -85,B 0,C 180,E1 -20250,E2 -20250} C_VEL
LIN {X 0,Y 218.472,Z 628.745,A -85,B 0,C 180,E1 -20251.844,E2 -20251.844} C_VEL
LIN {X 0,Y 218.482,Z 626.751,A -85,B 0,C 180,E1 -20254.292,E2 -20254.292} C_VEL
LIN {X 0,Y 218.76,Z 623.134,A -85,B 0,C 180,E1 -20257.384,E2 -20257.384} C_VEL
LIN {X 0,Y 219.322,Z 618.739,A -85,B 0,C 180,E1 -20260.151,E2 -20260.151} C_VEL
LIN {X 0,Y 220.182,Z 613.124,A -85,B 0,C 180,E1 -20262.911,E2 -20262.911} C_VEL
LIN {X 0,Y 221.528,Z 606.096,A -85,B 0,C 180,E1 -20265.644,E2 -20265.644} C_VEL
LIN {X 0,Y 223.321,Z 597.264,A -85,B 0,C 180,E1 -20268.343,E2 -20268.343} C_VEL
LIN {X 0,Y 225.12,Z 587.188,A -85,B 0,C 180,E1 -20270.801,E2 -20270.801} C_VEL
LIN {X 0,Y 226.962,Z 576.89,A -85,B 0,C 180,E1 -20272.772,E2 -20272.772} C_VEL
LIN {X 0,Y 228.923,Z 565.458,A -85,B 0,C 180,E1 -20274.485,E2 -20274.485} C_VEL
LIN {X 0,Y 230.69,Z 553.575,A -85,B 0,C 180,E1 -20275.851,E2 -20275.851} C_VEL
LIN {X 0,Y 232.005,Z 541.166,A -85,B 0,C 180,E1 -20276.904,E2 -20276.904} C_VEL
LIN {X 0,Y 233.121,Z 527.385,A -85,B 0,C 180,E1 -20277.675,E2 -20277.675} C_VEL
LIN {X 0,Y 235.129,Z 466.191,A -85,B 0,C 180,E1 -20279.549,E2 -20279.549} C_VEL
LIN {X 0,Y 232.237,Z 444.265,A -85,B 0,C 180,E1 -20280.618,E2 -20280.618} C_VEL
LIN {X 0,Y 226.638,Z 428.928,A -85,B 0,C 180,E1 -20281.827,E2 -20281.827} C_VEL
LIN {X 0,Y 222.59,Z 419.149,A -85,B 0,C 180,E1 -20282.738,E2 -20282.738} C_VEL
LIN {X 0,Y 222.338,Z 418.069,A -85,B 0,C 180,E1 -20283.042,E2 -20283.042} C_VEL
LIN {X 0,Y 220.878,Z 411.503,A -85,B 0,C 180,E1 -20286.201,E2 -20286.201} C_VEL
LIN {X 0,Y 220.808,Z 411.469,A -85,B 0,C 180,E1 -20290.192,E2 -20290.192} C_VEL
LIN {X 0,Y 220.829,Z 411.444,A -85,B 0,C 180,E1 -20294.439,E2 -20294.439} C_VEL
LIN {X 0,Y 220.853,Z 411.448,A -85,B 0,C 180,E1 -20298.067,E2 -20298.067} C_VEL
LIN {X 0,Y 220.838,Z 411.471,A -85,B 0,C 180,E1 -20302.712,E2 -20302.712} C_VEL
LIN {X 0,Y 220.822,Z 411.481,A -85,B 0,C 180,E1 -20307.245,E2 -20307.245} C_VEL
LIN {X 0,Y 220.826,Z 411.461,A -85,B 0,C 180,E1 -20311.485,E2 -20311.485} C_VEL
LIN {X 0,Y 220.861,Z 411.475,A -85,B 0,C 180,E1 -20315.564,E2 -20315.564} C_VEL
LIN {X 0,Y 220.882,Z 411.448,A -85,B 0,C 180,E1 -20319.513,E2 -20319.513} C_VEL
LIN {X 0,Y 221.014,Z 411.453,A -85,B 0,C 180,E1 -20323.37,E2 -20323.37} C_VEL
LIN {X 0,Y 221.008,Z 411.444,A -85,B 0,C 180,E1 -20327.138,E2 -20327.138} C_VEL
LIN {X 0,Y 221.202,Z 411.408,A -85,B 0,C 180,E1 -20330.859,E2 -20330.859} C_VEL
LIN {X 0,Y 221.257,Z 411.416,A -85,B 0,C 180,E1 -20332.7,E2 -20332.7} C_VEL
LIN {X 0,Y 221.51,Z 411.382,A -85,B 0,C 180,E1 -20338.182,E2 -20338.182} C_VEL
LIN {X 0,Y 221.51,Z 411.365,A -85,B 0,C 180,E1 -20341.818,E2 -20341.818} C_VEL
LIN {X 0,Y 221.269,Z 411.423,A -85,B 0,C 180,E1 -20347.299,E2 -20347.299} C_VEL
LIN {X 0,Y 221.065,Z 411.423,A -85,B 0,C 180,E1 -20350.996,E2 -20350.996} C_VEL
LIN {X 0,Y 221.014,Z 411.449,A -85,B 0,C 180,E1 -20356.63,E2 -20356.63} C_VEL
LIN {X 0,Y 220.89,Z 411.464,A -85,B 0,C 180,E1 -20360.486,E2 -20360.486} C_VEL
LIN {X 0,Y 220.865,Z 411.446,A -85,B 0,C 180,E1 -20364.435,E2 -20364.435} C_VEL
LIN {X 0,Y 220.835,Z 411.474,A -85,B 0,C 180,E1 -20368.514,E2 -20368.514} C_VEL
LIN {X 0,Y 220.816,Z 411.457,A -85,B 0,C 180,E1 -20372.756,E2 -20372.756} C_VEL
LIN {X 0,Y 220.809,Z 411.48,A -85,B 0,C 180,E1 -20377.279,E2 -20377.279} C_VEL
LIN {X 0,Y 220.77,Z 411.464,A -85,B 0,C 180,E1 -20381.953,E2 -20381.953} C_VEL
LIN {X 0,Y 220.852,Z 411.472,A -85,B 0,C 180,E1 -20387.047,E2 -20387.047} C_VEL
LIN {X 0,Y 220.85,Z 411.47,A -85,B 0,C 180,E1 -20390.473,E2 -20390.473} C_VEL
LIN {X 0,Y 220.816,Z 411.459,A -85,B 0,C 180,E1 -20395.048,E2 -20395.048} C_VEL
LIN {X 0,Y 220.869,Z 411.448,A -85,B 0,C 180,E1 -20399.395,E2 -20399.395} C_VEL
LIN {X 0,Y 220.896,Z 411.451,A -85,B 0,C 180,E1 -20403.55,E2 -20403.55} C_VEL
LIN {X 0,Y 220.951,Z 411.479,A -85,B 0,C 180,E1 -20409.032,E2 -20409.032} C_VEL
LIN {X 0,Y 221.059,Z 412.067,A -85,B 0,C 180,E1 -20409.53,E2 -20409.53} C_VEL
LIN {X 0,Y 221.51,Z 413.822,A -85,B 0,C 180,E1 -20410.179,E2 -20410.179} C_VEL
LIN {X 0,Y 228.873,Z 431.219,A -85,B 0,C 180,E1 -20411.785,E2 -20411.785} C_VEL
LIN {X 0,Y 234.051,Z 446.199,A -85,B 0,C 180,E1 -20412.915,E2 -20412.915} C_VEL
LIN {X 0,Y 235.525,Z 457.317,A -85,B 0,C 180,E1 -20413.455,E2 -20413.455} C_VEL
LIN {X 0,Y 233.22,Z 520.594,A -85,B 0,C 180,E1 -20415.352,E2 -20415.352} C_VEL
LIN {X 0,Y 232.256,Z 533.698,A -85,B 0,C 180,E1 -20416.067,E2 -20416.067} C_VEL
LIN {X 0,Y 230.89,Z 546.742,A -85,B 0,C 180,E1 -20417.138,E2 -20417.138} C_VEL
LIN {X 0,Y 229.323,Z 558.125,A -85,B 0,C 180,E1 -20418.42,E2 -20418.42} C_VEL
LIN {X 0,Y 227.471,Z 568.959,A -85,B 0,C 180,E1 -20419.991,E2 -20419.991} C_VEL
LIN {X 0,Y 225.777,Z 578.442,A -85,B 0,C 180,E1 -20421.722,E2 -20421.722} C_VEL
LIN {X 0,Y 223.752,Z 589.03,A -85,B 0,C 180,E1 -20424.141,E2 -20424.141} C_VEL
LIN {X 0,Y 222.019,Z 598.168,A -85,B 0,C 180,E1 -20426.824,E2 -20426.824} C_VEL
LIN {X 0,Y 220.621,Z 605.54,A -85,B 0,C 180,E1 -20429.543,E2 -20429.543} C_VEL
LIN {X 0,Y 219.706,Z 610.542,A -85,B 0,C 180,E1 -20431.833,E2 -20431.833} C_VEL
LIN {X 0,Y 219.078,Z 615.388,A -85,B 0,C 180,E1 -20434.599,E2 -20434.599} C_VEL
LIN {X 0,Y 218.576,Z 619.125,A -85,B 0,C 180,E1 -20437.389,E2 -20437.389} C_VEL
LIN {X 0,Y 218.321,Z 621.06,A -85,B 0,C 180,E1 -20439.262,E2 -20439.262} C_VEL
LIN {X 0,Y 218.184,Z 622.533,A -85,B 0,C 180,E1 -20441.143,E2 -20441.143} C_VEL
LIN {X 0,Y 218.197,Z 623.571,A -85,B 0,C 180,E1 -20443.03,E2 -20443.03} C_VEL
LIN {X 0,Y 218.278,Z 624.232,A -85,B 0,C 180,E1 -20445,E2 -20445} C_VEL
LIN {X 0,Y 218.384,Z 624.453,A -85,B 0,C 180,E1 -20446.835,E2 -20446.835} C_VEL
LIN {X 0,Y 218.628,Z 624.235,A -85,B 0,C 180,E1 -20448.75,E2 -20448.75} C_VEL
LIN {X 0,Y 219.371,Z 623.091,A -85,B 0,C 180,E1 -20451.709,E2 -20451.709} C_VEL
LIN {X 0,Y 220.407,Z 621.071,A -85,B 0,C 180,E1 -20454.488,E2 -20454.488} C_VEL
LIN {X 0,Y 222.097,Z 617.563,A -85,B 0,C 180,E1 -20457.622,E2 -20457.622} C_VEL
LIN {X 0,Y 224.683,Z 612.026,A -85,B 0,C 180,E1 -20461.071,E2 -20461.071} C_VEL
LIN {X 0,Y 227.285,Z 606.035,A -85,B 0,C 180,E1 -20463.819,E2 -20463.819} C_VEL
LIN {X 0,Y 230.402,Z 598.479,A -85,B 0,C 180,E1 -20466.498,E2 -20466.498} C_VEL
LIN {X 0,Y 233.59,Z 590.163,A -85,B 0,C 180,E1 -20468.816,E2 -20468.816} C_VEL
LIN {X 0,Y 236.763,Z 581.298,A -85,B 0,C 180,E1 -20470.77,E2 -20470.77} C_VEL
LIN {X 0,Y 239.61,Z 572.019,A -85,B 0,C 180,E1 -20472.422,E2 -20472.422} C_VEL
LIN {X 0,Y 242.639,Z 560.449,A -85,B 0,C 180,E1 -20474.038,E2 -20474.038} C_VEL
LIN {X 0,Y 245.198,Z 548.384,A -85,B 0,C 180,E1 -20475.33,E2 -20475.33} C_VEL
LIN {X 0,Y 247.349,Z 535.932,A -85,B 0,C 180,E1 -20476.281,E2 -20476.281} C_VEL
LIN {X 0,Y 248.841,Z 523.072,A -85,B 0,C 180,E1 -20476.95,E2 -20476.95} C_VEL
LIN {X 0,Y 250.111,Z 502.147,A -85,B 0,C 180,E1 -20477.58,E2 -20477.58} C_VEL
LIN {X 0,Y 251.842,Z 467.934,A -85,B 0,C 180,E1 -20478.516,E2 -20478.516} C_VEL
LIN {X 0,Y 245.258,Z 453.377,A -85,B 0,C 180,E1 -20480.421,E2 -20480.421} C_VEL
LIN {X 0,Y 238.712,Z 441.055,A -85,B 0,C 180,E1 -20482.409,E2 -20482.409} C_VEL
LIN {X 0,Y 231.604,Z 429.042,A -85,B 0,C 180,E1 -20484.733,E2 -20484.733} C_VEL
LIN {X 0,Y 227.943,Z 423.559,A -85,B 0,C 180,E1 -20485.996,E2 -20485.996} C_VEL
LIN {X 0,Y 224.278,Z 418.362,A -85,B 0,C 180,E1 -20487.323,E2 -20487.323} C_VEL
LIN {X 0,Y 221.718,Z 414.327,A -85,B 0,C 180,E1 -20488.4,E2 -20488.4} C_VEL
LIN {X 0,Y 220.89,Z 411.72,A -85,B 0,C 180,E1 -20490.189,E2 -20490.189} C_VEL
LIN {X 0,Y 220.823,Z 411.457,A -85,B 0,C 180,E1 -20491.485,E2 -20491.485} C_VEL
LIN {X 0,Y 220.862,Z 411.47,A -85,B 0,C 180,E1 -20495.565,E2 -20495.565} C_VEL
LIN {X 0,Y 220.888,Z 411.471,A -85,B 0,C 180,E1 -20499.514,E2 -20499.514} C_VEL
LIN {X 0,Y 221.011,Z 411.456,A -85,B 0,C 180,E1 -20503.37,E2 -20503.37} C_VEL
LIN {X 0,Y 221.107,Z 411.432,A -85,B 0,C 180,E1 -20509.006,E2 -20509.006} C_VEL
LIN {X 0,Y 221.301,Z 411.415,A -85,B 0,C 180,E1 -20512.702,E2 -20512.702} C_VEL
LIN {X 0,Y 221.519,Z 411.38,A -85,B 0,C 180,E1 -20518.182,E2 -20518.182} C_VEL
LIN {X 0,Y 221.509,Z 411.393,A -85,B 0,C 180,E1 -20521.818,E2 -20521.818} C_VEL
LIN {X 0,Y 221.284,Z 411.416,A -85,B 0,C 180,E1 -20527.299,E2 -20527.299} C_VEL
LIN {X 0,Y 221.107,Z 411.443,A -85,B 0,C 180,E1 -20530.995,E2 -20530.995} C_VEL
LIN {X 0,Y 221.011,Z 411.452,A -85,B 0,C 180,E1 -20536.63,E2 -20536.63} C_VEL
LIN {X 0,Y 220.888,Z 411.471,A -85,B 0,C 180,E1 -20540.487,E2 -20540.487} C_VEL
LIN {X 0,Y 220.863,Z 411.472,A -85,B 0,C 180,E1 -20544.436,E2 -20544.436} C_VEL
LIN {X 0,Y 220.833,Z 411.477,A -85,B 0,C 180,E1 -20548.514,E2 -20548.514} C_VEL
LIN {X 0,Y 220.806,Z 411.475,A -85,B 0,C 180,E1 -20552.294,E2 -20552.294} C_VEL
LIN {X 0,Y 220.134,Z 411.565,A -85,B 0,C 180,E1 -20553.307,E2 -20553.307} C_VEL
LIN {X 0,Y 217.275,Z 411.921,A -85,B 0,C 180,E1 -20554.898,E2 -20554.898} C_VEL
LIN {X 0,Y 214.412,Z 412.274,A -85,B 0,C 180,E1 -20556.53,E2 -20556.53} C_VEL
LIN {X 0,Y 213.776,Z 412.351,A -85,B 0,C 180,E1 -20557.589,E2 -20557.589} C_VEL
LIN {X 0,Y 213.815,Z 412.553,A -85,B 0,C 180,E1 -20558.422,E2 -20558.422} C_VEL
LIN {X 0,Y 215.44,Z 417.825,A -85,B 0,C 180,E1 -20562.522,E2 -20562.522} C_VEL
LIN {X 0,Y 218.539,Z 422.697,A -85,B 0,C 180,E1 -20563.94,E2 -20563.94} C_VEL
LIN {X 0,Y 223.479,Z 430.106,A -85,B 0,C 180,E1 -20565.867,E2 -20565.867} C_VEL
LIN {X 0,Y 229.434,Z 439.737,A -85,B 0,C 180,E1 -20568.023,E2 -20568.023} C_VEL
LIN {X 0,Y 235.594,Z 450.896,A -85,B 0,C 180,E1 -20570.108,E2 -20570.108} C_VEL
LIN {X 0,Y 241.742,Z 463.615,A -85,B 0,C 180,E1 -20572.071,E2 -20572.071} C_VEL
LIN {X 0,Y 245.951,Z 473.585,A -85,B 0,C 180,E1 -20573.366,E2 -20573.366} C_VEL
LIN {X 0,Y 246.018,Z 478.572,A -85,B 0,C 180,E1 -20573.572,E2 -20573.572} C_VEL
LIN {X 0,Y 243.41,Z 526.081,A -85,B 0,C 180,E1 -20574.919,E2 -20574.919} C_VEL
LIN {X 0,Y 241.915,Z 539.195,A -85,B 0,C 180,E1 -20575.558,E2 -20575.558} C_VEL
LIN {X 0,Y 239.682,Z 552.385,A -85,B 0,C 180,E1 -20576.523,E2 -20576.523} C_VEL
LIN {X 0,Y 236.882,Z 564.307,A -85,B 0,C 180,E1 -20577.723,E2 -20577.723} C_VEL
LIN {X 0,Y 233.829,Z 575.683,A -85,B 0,C 180,E1 -20579.274,E2 -20579.274} C_VEL
LIN {X 0,Y 230.523,Z 585.967,A -85,B 0,C 180,E1 -20581.055,E2 -20581.055} C_VEL
LIN {X 0,Y 227.466,Z 594.391,A -85,B 0,C 180,E1 -20582.889,E2 -20582.889} C_VEL
LIN {X 0,Y 224.361,Z 602.181,A -85,B 0,C 180,E1 -20584.984,E2 -20584.984} C_VEL
LIN {X 0,Y 221.162,Z 609.806,A -85,B 0,C 180,E1 -20587.585,E2 -20587.585} C_VEL
LIN {X 0,Y 218.418,Z 615.951,A -85,B 0,C 180,E1 -20590.255,E2 -20590.255} C_VEL
LIN {X 0,Y 216.011,Z 620.855,A -85,B 0,C 180,E1 -20592.974,E2 -20592.974} C_VEL
LIN {X 0,Y 214.265,Z 624.653,A -85,B 0,C 180,E1 -20595.76,E2 -20595.76} C_VEL
LIN {X 0,Y 212.904,Z 627.456,A -85,B 0,C 180,E1 -20598.577,E2 -20598.577} C_VEL
LIN {X 0,Y 211.833,Z 629.738,A -85,B 0,C 180,E1 -20602.375,E2 -20602.375} C_VEL
LIN {X 0,Y 211.425,Z 630.456,A -85,B 0,C 180,E1 -20605.74,E2 -20605.74} C_VEL
LIN {X 0,Y 211.38,Z 630.204,A -85,B 0,C 180,E1 -20608.095,E2 -20608.095} C_VEL
LIN {X 0,Y 211.458,Z 629.573,A -85,B 0,C 180,E1 -20610,E2 -20610} C_VEL
LIN {X 0,Y 211.377,Z 628.546,A -85,B 0,C 180,E1 -20611.906,E2 -20611.906} C_VEL
LIN {X 0,Y 211.389,Z 626.788,A -85,B 0,C 180,E1 -20614.124,E2 -20614.124} C_VEL
LIN {X 0,Y 211.689,Z 622.816,A -85,B 0,C 180,E1 -20617.632,E2 -20617.632} C_VEL
LIN {X 0,Y 212.308,Z 618.357,A -85,B 0,C 180,E1 -20620.49,E2 -20620.49} C_VEL
LIN {X 0,Y 213.208,Z 612.67,A -85,B 0,C 180,E1 -20623.341,E2 -20623.341} C_VEL
LIN {X 0,Y 214.664,Z 605.527,A -85,B 0,C 180,E1 -20626.158,E2 -20626.158} C_VEL
LIN {X 0,Y 216.573,Z 596.596,A -85,B 0,C 180,E1 -20628.936,E2 -20628.936} C_VEL
LIN {X 0,Y 218.238,Z 587.391,A -85,B 0,C 180,E1 -20631.241,E2 -20631.241} C_VEL
LIN {X 0,Y 220.15,Z 577.19,A -85,B 0,C 180,E1 -20633.269,E2 -20633.269} C_VEL
LIN {X 0,Y 222.174,Z 565.848,A -85,B 0,C 180,E1 -20635.03,E2 -20635.03} C_VEL
LIN {X 0,Y 223.995,Z 554.09,A -85,B 0,C 180,E1 -20636.432,E2 -20636.432} C_VEL
LIN {X 0,Y 225.421,Z 541.235,A -85,B 0,C 180,E1 -20637.567,E2 -20637.567} C_VEL
LIN {X 0,Y 226.556,Z 527.918,A -85,B 0,C 180,E1 -20638.339,E2 -20638.339} C_VEL
LIN {X 0,Y 227.869,Z 494.235,A -85,B 0,C 180,E1 -20639.419,E2 -20639.419} C_VEL
LIN {X 0,Y 228.657,Z 466.723,A -85,B 0,C 180,E1 -20640.273,E2 -20640.273} C_VEL
LIN {X 0,Y 226.04,Z 446.516,A -85,B 0,C 180,E1 -20641.29,E2 -20641.29} C_VEL
LIN {X 0,Y 220.612,Z 431.678,A -85,B 0,C 180,E1 -20642.519,E2 -20642.519} C_VEL
LIN {X 0,Y 215.314,Z 418.776,A -85,B 0,C 180,E1 -20643.794,E2 -20643.794} C_VEL
LIN {X 0,Y 214.426,Z 415.04,A -85,B 0,C 180,E1 -20645.466,E2 -20645.466} C_VEL
LIN {X 0,Y 213.827,Z 412.392,A -85,B 0,C 180,E1 -20646.84,E2 -20646.84} C_VEL
LIN {X 0,Y 213.754,Z 412.357,A -85,B 0,C 180,E1 -20651.115,E2 -20651.115} C_VEL
LIN {X 0,Y 213.809,Z 412.328,A -85,B 0,C 180,E1 -20653.685,E2 -20653.685} C_VEL
LIN {X 0,Y 213.812,Z 412.306,A -85,B 0,C 180,E1 -20656.348,E2 -20656.348} C_VEL
LIN {X 0,Y 213.795,Z 412.343,A -85,B 0,C 180,E1 -20659.118,E2 -20659.118} C_VEL
LIN {X 0,Y 213.754,Z 412.345,A -85,B 0,C 180,E1 -20663.713,E2 -20663.713} C_VEL
LIN {X 0,Y 213.769,Z 412.357,A -85,B 0,C 180,E1 -20668.262,E2 -20668.262} C_VEL
LIN {X 0,Y 213.825,Z 412.339,A -85,B 0,C 180,E1 -20672.603,E2 -20672.603} C_VEL
LIN {X 0,Y 213.818,Z 412.346,A -85,B 0,C 180,E1 -20676.973,E2 -20676.973} C_VEL
LIN {X 0,Y 213.942,Z 412.33,A -85,B 0,C 180,E1 -20682.803,E2 -20682.803} C_VEL
LIN {X 0,Y 213.95,Z 412.327,A -85,B 0,C 180,E1 -20686.706,E2 -20686.706} C_VEL
LIN {X 0,Y 214.14,Z 412.284,A -85,B 0,C 180,E1 -20690.555,E2 -20690.555} C_VEL
LIN {X 0,Y 214.099,Z 412.314,A -85,B 0,C 180,E1 -20694.348,E2 -20694.348} C_VEL
LIN {X 0,Y 214.443,Z 412.262,A -85,B 0,C 180,E1 -20698.122,E2 -20698.122} C_VEL
LIN {X 0,Y 214.548,Z 412.23,A -85,B 0,C 180,E1 -20700,E2 -20700} C_VEL
LIN {X 0,Y 214.443,Z 412.244,A -85,B 0,C 180,E1 -20701.878,E2 -20701.878} C_VEL
LIN {X 0,Y 214.206,Z 412.301,A -85,B 0,C 180,E1 -20707.541,E2 -20707.541} C_VEL
LIN {X 0,Y 213.997,Z 412.299,A -85,B 0,C 180,E1 -20711.364,E2 -20711.364} C_VEL
LIN {X 0,Y 213.929,Z 412.323,A -85,B 0,C 180,E1 -20715.237,E2 -20715.237} C_VEL
LIN {X 0,Y 213.838,Z 412.347,A -85,B 0,C 180,E1 -20719.187,E2 -20719.187} C_VEL
LIN {X 0,Y 213.846,Z 412.317,A -85,B 0,C 180,E1 -20723.227,E2 -20723.227} C_VEL
LIN {X 0,Y 213.828,Z 412.346,A -85,B 0,C 180,E1 -20727.45,E2 -20727.45} C_VEL
LIN {X 0,Y 213.776,Z 412.342,A -85,B 0,C 180,E1 -20731.736,E2 -20731.736} C_VEL
LIN {X 0,Y 213.742,Z 412.354,A -85,B 0,C 180,E1 -20736.288,E2 -20736.288} C_VEL
LIN {X 0,Y 213.711,Z 412.346,A -85,B 0,C 180,E1 -20741.125,E2 -20741.125} C_VEL
LIN {X 0,Y 213.776,Z 412.356,A -85,B 0,C 180,E1 -20746.34,E2 -20746.34} C_VEL
LIN {X 0,Y 213.786,Z 412.342,A -85,B 0,C 180,E1 -20749.122,E2 -20749.122} C_VEL
LIN {X 0,Y 213.755,Z 412.355,A -85,B 0,C 180,E1 -20753.714,E2 -20753.714} C_VEL
LIN {X 0,Y 213.796,Z 412.317,A -85,B 0,C 180,E1 -20758.725,E2 -20758.725} C_VEL
LIN {X 0,Y 213.827,Z 412.343,A -85,B 0,C 180,E1 -20762.603,E2 -20762.603} C_VEL
LIN {X 0,Y 213.849,Z 412.344,A -85,B 0,C 180,E1 -20767.794,E2 -20767.794} C_VEL
LIN {X 0,Y 213.943,Z 412.654,A -85,B 0,C 180,E1 -20768.691,E2 -20768.691} C_VEL
LIN {X 0,Y 214.305,Z 414.039,A -85,B 0,C 180,E1 -20769.167,E2 -20769.167} C_VEL
LIN {X 0,Y 221.219,Z 429.851,A -85,B 0,C 180,E1 -20770.752,E2 -20770.752} C_VEL
LIN {X 0,Y 227.176,Z 446.145,A -85,B 0,C 180,E1 -20772.093,E2 -20772.093} C_VEL
LIN {X 0,Y 228.232,Z 450.951,A -85,B 0,C 180,E1 -20772.388,E2 -20772.388} C_VEL
LIN {X 0,Y 229.051,Z 458.553,A -85,B 0,C 180,E1 -20772.748,E2 -20772.748} C_VEL
LIN {X 0,Y 226.693,Z 520.65,A -85,B 0,C 180,E1 -20774.655,E2 -20774.655} C_VEL
LIN {X 0,Y 225.689,Z 534.152,A -85,B 0,C 180,E1 -20775.418,E2 -20775.418} C_VEL
LIN {X 0,Y 224.272,Z 546.864,A -85,B 0,C 180,E1 -20776.49,E2 -20776.49} C_VEL
LIN {X 0,Y 222.535,Z 559.072,A -85,B 0,C 180,E1 -20777.922,E2 -20777.922} C_VEL
LIN {X 0,Y 220.502,Z 570.53,A -85,B 0,C 180,E1 -20779.672,E2 -20779.672} C_VEL
LIN {X 0,Y 218.795,Z 579.757,A -85,B 0,C 180,E1 -20781.456,E2 -20781.456} C_VEL
LIN {X 0,Y 217.032,Z 588.369,A -85,B 0,C 180,E1 -20783.492,E2 -20783.492} C_VEL
LIN {X 0,Y 215.507,Z 596.284,A -85,B 0,C 180,E1 -20785.792,E2 -20785.792} C_VEL
LIN {X 0,Y 213.861,Z 604.041,A -85,B 0,C 180,E1 -20788.587,E2 -20788.587} C_VEL
LIN {X 0,Y 212.937,Z 609.331,A -85,B 0,C 180,E1 -20790.945,E2 -20790.945} C_VEL
LIN {X 0,Y 212.15,Z 614.46,A -85,B 0,C 180,E1 -20793.798,E2 -20793.798} C_VEL
LIN {X 0,Y 211.588,Z 618.451,A -85,B 0,C 180,E1 -20796.675,E2 -20796.675} C_VEL
LIN {X 0,Y 211.18,Z 621.404,A -85,B 0,C 180,E1 -20799.578,E2 -20799.578} C_VEL
LIN {X 0,Y 211.076,Z 622.799,A -85,B 0,C 180,E1 -20801.523,E2 -20801.523} C_VEL
LIN {X 0,Y 211.18,Z 624.32,A -85,B 0,C 180,E1 -20805.179,E2 -20805.179} C_VEL
LIN {X 0,Y 211.357,Z 624.539,A -85,B 0,C 180,E1 -20807.413,E2 -20807.413} C_VEL
LIN {X 0,Y 211.652,Z 624.267,A -85,B 0,C 180,E1 -20809.393,E2 -20809.393} C_VEL
LIN {X 0,Y 212.399,Z 623.226,A -85,B 0,C 180,E1 -20812.107,E2 -20812.107} C_VEL
LIN {X 0,Y 213.654,Z 620.908,A -85,B 0,C 180,E1 -20815.316,E2 -20815.316} C_VEL
LIN {X 0,Y 215.276,Z 617.774,A -85,B 0,C 180,E1 -20818.182,E2 -20818.182} C_VEL
LIN {X 0,Y 217.507,Z 613.326,A -85,B 0,C 180,E1 -20821.129,E2 -20821.129} C_VEL
LIN {X 0,Y 220.467,Z 607.013,A -85,B 0,C 180,E1 -20824.261,E2 -20824.261} C_VEL
LIN {X 0,Y 223.334,Z 600.577,A -85,B 0,C 180,E1 -20826.718,E2 -20826.718} C_VEL
LIN {X 0,Y 226.63,Z 592.457,A -85,B 0,C 180,E1 -20829.17,E2 -20829.17} C_VEL
LIN {X 0,Y 230.467,Z 582.285,A -85,B 0,C 180,E1 -20831.547,E2 -20831.547} C_VEL
LIN {X 0,Y 233.817,Z 571.961,A -85,B 0,C 180,E1 -20833.436,E2 -20833.436} C_VEL
LIN {X 0,Y 237.017,Z 560.162,A -85,B 0,C 180,E1 -20835.1,E2 -20835.1} C_VEL
LIN {X 0,Y 239.652,Z 548.243,A -85,B 0,C 180,E1 -20836.382,E2 -20836.382} C_VEL
LIN {X 0,Y 241.886,Z 535.667,A -85,B 0,C 180,E1 -20837.344,E2 -20837.344} C_VEL
LIN {X 0,Y 243.447,Z 522.644,A -85,B 0,C 180,E1 -20838.017,E2 -20838.017} C_VEL
LIN {X 0,Y 245.026,Z 496.108,A -85,B 0,C 180,E1 -20838.806,E2 -20838.806} C_VEL
LIN {X 0,Y 246.357,Z 470.198,A -85,B 0,C 180,E1 -20839.533,E2 -20839.533} C_VEL
LIN {X 0,Y 240.462,Z 457,A -85,B 0,C 180,E1 -20841.338,E2 -20841.338} C_VEL
LIN {X 0,Y 234.113,Z 444.968,A -85,B 0,C 180,E1 -20843.37,E2 -20843.37} C_VEL
LIN {X 0,Y 227.814,Z 434.121,A -85,B 0,C 180,E1 -20845.535,E2 -20845.535} C_VEL
LIN {X 0,Y 221.565,Z 424.701,A -85,B 0,C 180,E1 -20847.839,E2 -20847.839} C_VEL
LIN {X 0,Y 217.456,Z 418.983,A -85,B 0,C 180,E1 -20849.468,E2 -20849.468} C_VEL
LIN {X 0,Y 214.338,Z 414.311,A -85,B 0,C 180,E1 -20850.943,E2 -20850.943} C_VEL
LIN {X 0,Y 213.825,Z 412.371,A -85,B 0,C 180,E1 -20852.55,E2 -20852.55} C_VEL
LIN {X 0,Y 213.847,Z 412.343,A -85,B 0,C 180,E1 -20856.952,E2 -20856.952} C_VEL
LIN {X 0,Y 213.938,Z 412.331,A -85,B 0,C 180,E1 -20862.803,E2 -20862.803} C_VEL
LIN {X 0,Y 213.974,Z 412.324,A -85,B 0,C 180,E1 -20866.708,E2 -20866.708} C_VEL
LIN {X 0,Y 214.162,Z 412.296,A -85,B 0,C 180,E1 -20870.556,E2 -20870.556} C_VEL
LIN {X 0,Y 214.235,Z 412.298,A -85,B 0,C 180,E1 -20872.46,E2 -20872.46} C_VEL
LIN {X 0,Y 214.476,Z 412.258,A -85,B 0,C 180,E1 -20878.122,E2 -20878.122} C_VEL
LIN {X 0,Y 214.549,Z 412.248,A -85,B 0,C 180,E1 -20880,E2 -20880} C_VEL
LIN {X 0,Y 214.442,Z 412.274,A -85,B 0,C 180,E1 -20881.878,E2 -20881.878} C_VEL
LIN {X 0,Y 214.222,Z 412.292,A -85,B 0,C 180,E1 -20887.541,E2 -20887.541} C_VEL
LIN {X 0,Y 214.04,Z 412.324,A -85,B 0,C 180,E1 -20891.362,E2 -20891.362} C_VEL
LIN {X 0,Y 213.929,Z 412.332,A -85,B 0,C 180,E1 -20895.237,E2 -20895.237} C_VEL
LIN {X 0,Y 213.835,Z 412.337,A -85,B 0,C 180,E1 -20899.188,E2 -20899.188} C_VEL
LIN {X 0,Y 213.843,Z 412.335,A -85,B 0,C 180,E1 -20903.228,E2 -20903.228} C_VEL
LIN {X 0,Y 213.825,Z 412.34,A -85,B 0,C 180,E1 -20907.451,E2 -20907.451} C_VEL
LIN {X 0,Y 213.744,Z 412.351,A -85,B 0,C 180,E1 -20912.273,E2 -20912.273} C_VEL
LIN {X 0,Y 213.756,Z 412.356,A -85,B 0,C 180,E1 -20916.286,E2 -20916.286} C_VEL
LIN {X 0,Y 213.776,Z 412.351,A -85,B 0,C 180,E1 -20917.589,E2 -20917.589} C_VEL
LIN {X 0,Y 213.79,Z 413.017,A -85,B 0,C 180,E1 -20918.597,E2 -20918.597} C_VEL
LIN {X 0,Y 213.767,Z 415.232,A -85,B 0,C 180,E1 -20919.751,E2 -20919.751} C_VEL
LIN {X 0,Y 213.911,Z 419.803,A -85,B 0,C 180,E1 -20921.148,E2 -20921.148} C_VEL
LIN {X 0,Y 215.291,Z 427.6,A -85,B 0,C 180,E1 -20922.957,E2 -20922.957} C_VEL
LIN {X 0,Y 217.442,Z 431.678,A -85,B 0,C 180,E1 -20924.05,E2 -20924.05} C_VEL
LIN {X 0,Y 220.344,Z 436.095,A -85,B 0,C 180,E1 -20925.207,E2 -20925.207} C_VEL
LIN {X 0,Y 225.578,Z 444.666,A -85,B 0,C 180,E1 -20927.184,E2 -20927.184} C_VEL
LIN {X 0,Y 231.52,Z 455.683,A -85,B 0,C 180,E1 -20929.295,E2 -20929.295} C_VEL
LIN {X 0,Y 237.729,Z 468.851,A -85,B 0,C 180,E1 -20931.376,E2 -20931.376} C_VEL
LIN {X 0,Y 240.759,Z 476.057,A -85,B 0,C 180,E1 -20932.355,E2 -20932.355} C_VEL
LIN {X 0,Y 238.049,Z 525.869,A -85,B 0,C 180,E1 -20933.811,E2 -20933.811} C_VEL
LIN {X 0,Y 236.493,Z 539.017,A -85,B 0,C 180,E1 -20934.456,E2 -20934.456} C_VEL
LIN {X 0,Y 234.293,Z 551.662,A -85,B 0,C 180,E1 -20935.386,E2 -20935.386} C_VEL
LIN {X 0,Y 231.394,Z 563.764,A -85,B 0,C 180,E1 -20936.6,E2 -20936.6} C_VEL
LIN {X 0,Y 228.593,Z 573.943,A -85,B 0,C 180,E1 -20937.973,E2 -20937.973} C_VEL
LIN {X 0,Y 225.126,Z 584.508,A -85,B 0,C 180,E1 -20939.777,E2 -20939.777} C_VEL
LIN {X 0,Y 221.206,Z 594.91,A -85,B 0,C 180,E1 -20942.056,E2 -20942.056} C_VEL
LIN {X 0,Y 217.954,Z 602.587,A -85,B 0,C 180,E1 -20944.196,E2 -20944.196} C_VEL
LIN {X 0,Y 214.622,Z 610.106,A -85,B 0,C 180,E1 -20946.863,E2 -20946.863} C_VEL
LIN {X 0,Y 211.76,Z 616.175,A -85,B 0,C 180,E1 -20949.607,E2 -20949.607} C_VEL
LIN {X 0,Y 209.238,Z 621.01,A -85,B 0,C 180,E1 -20952.405,E2 -20952.405} C_VEL
LIN {X 0,Y 207.356,Z 624.744,A -85,B 0,C 180,E1 -20955.275,E2 -20955.275} C_VEL
LIN {X 0,Y 205.931,Z 627.485,A -85,B 0,C 180,E1 -20958.185,E2 -20958.185} C_VEL
LIN {X 0,Y 204.773,Z 629.709,A -85,B 0,C 180,E1 -20962.11,E2 -20962.11} C_VEL
LIN {X 0,Y 204.347,Z 630.354,A -85,B 0,C 180,E1 -20965.857,E2 -20965.857} C_VEL
LIN {X 0,Y 204.289,Z 630.062,A -85,B 0,C 180,E1 -20968.029,E2 -20968.029} C_VEL
LIN {X 0,Y 204.361,Z 629.402,A -85,B 0,C 180,E1 -20970,E2 -20970} C_VEL
LIN {X 0,Y 204.283,Z 628.342,A -85,B 0,C 180,E1 -20971.972,E2 -20971.972} C_VEL
LIN {X 0,Y 204.297,Z 626.825,A -85,B 0,C 180,E1 -20973.946,E2 -20973.946} C_VEL
LIN {X 0,Y 204.488,Z 623.751,A -85,B 0,C 180,E1 -20976.909,E2 -20976.909} C_VEL
LIN {X 0,Y 205.056,Z 619.603,A -85,B 0,C 180,E1 -20979.868,E2 -20979.868} C_VEL
LIN {X 0,Y 206.089,Z 613.235,A -85,B 0,C 180,E1 -20983.308,E2 -20983.308} C_VEL
LIN {X 0,Y 207.525,Z 606.287,A -85,B 0,C 180,E1 -20986.224,E2 -20986.224} C_VEL
LIN {X 0,Y 209.446,Z 597.563,A -85,B 0,C 180,E1 -20989.097,E2 -20989.097} C_VEL
LIN {X 0,Y 211.185,Z 588.571,A -85,B 0,C 180,E1 -20991.473,E2 -20991.473} C_VEL
LIN {X 0,Y 213.145,Z 578.689,A -85,B 0,C 180,E1 -20993.565,E2 -20993.565} C_VEL
LIN {X 0,Y 215.133,Z 567.801,A -85,B 0,C 180,E1 -20995.39,E2 -20995.39} C_VEL
LIN {X 0,Y 217.164,Z 555.571,A -85,B 0,C 180,E1 -20996.941,E2 -20996.941} C_VEL
LIN {X 0,Y 218.736,Z 542.721,A -85,B 0,C 180,E1 -20998.158,E2 -20998.158} C_VEL
LIN {X 0,Y 219.945,Z 529.777,A -85,B 0,C 180,E1 -20998.974,E2 -20998.974} C_VEL
LIN {X 0,Y 220.767,Z 511.612,A -85,B 0,C 180,E1 -20999.635,E2 -20999.635} C_VEL
LIN {X 0,Y 222.227,Z 467.39,A -85,B 0,C 180,E1 -21001.027,E2 -21001.027} C_VEL
LIN {X 0,Y 219.707,Z 448.218,A -85,B 0,C 180,E1 -21002.039,E2 -21002.039} C_VEL
LIN {X 0,Y 213.837,Z 432.315,A -85,B 0,C 180,E1 -21003.436,E2 -21003.436} C_VEL
LIN {X 0,Y 208.138,Z 419.019,A -85,B 0,C 180,E1 -21004.832,E2 -21004.832} C_VEL
LIN {X 0,Y 207.884,Z 418.05,A -85,B 0,C 180,E1 -21005.08,E2 -21005.08} C_VEL
LIN {X 0,Y 206.754,Z 413.28,A -85,B 0,C 180,E1 -21007.583,E2 -21007.583} C_VEL
LIN {X 0,Y 206.684,Z 413.23,A -85,B 0,C 180,E1 -21012.849,E2 -21012.849} C_VEL
LIN {X 0,Y 206.715,Z 413.193,A -85,B 0,C 180,E1 -21017.158,E2 -21017.158} C_VEL
LIN {X 0,Y 206.76,Z 413.232,A -85,B 0,C 180,E1 -21021.424,E2 -21021.424} C_VEL
LIN {X 0,Y 206.731,Z 413.22,A -85,B 0,C 180,E1 -21024.695,E2 -21024.695} C_VEL
LIN {X 0,Y 206.706,Z 413.23,A -85,B 0,C 180,E1 -21029.336,E2 -21029.336} C_VEL
LIN {X 0,Y 206.73,Z 413.23,A -85,B 0,C 180,E1 -21033.771,E2 -21033.771} C_VEL
LIN {X 0,Y 206.737,Z 413.219,A -85,B 0,C 180,E1 -21038.041,E2 -21038.041} C_VEL
LIN {X 0,Y 206.871,Z 413.208,A -85,B 0,C 180,E1 -21042.196,E2 -21042.196} C_VEL
LIN {X 0,Y 206.893,Z 413.208,A -85,B 0,C 180,E1 -21046.244,E2 -21046.244} C_VEL
LIN {X 0,Y 207.098,Z 413.157,A -85,B 0,C 180,E1 -21050.231,E2 -21050.231} C_VEL
LIN {X 0,Y 207.06,Z 413.191,A -85,B 0,C 180,E1 -21054.156,E2 -21054.156} C_VEL
LIN {X 0,Y 207.38,Z 413.141,A -85,B 0,C 180,E1 -21058.058,E2 -21058.058} C_VEL
LIN {X 0,Y 207.512,Z 413.104,A -85,B 0,C 180,E1 -21060,E2 -21060} C_VEL
LIN {X 0,Y 207.379,Z 413.122,A -85,B 0,C 180,E1 -21061.942,E2 -21061.942} C_VEL
LIN {X 0,Y 207.146,Z 413.179,A -85,B 0,C 180,E1 -21067.8,E2 -21067.8} C_VEL
LIN {X 0,Y 206.921,Z 413.175,A -85,B 0,C 180,E1 -21071.758,E2 -21071.758} C_VEL
LIN {X 0,Y 206.864,Z 413.207,A -85,B 0,C 180,E1 -21075.771,E2 -21075.771} C_VEL
LIN {X 0,Y 206.782,Z 413.222,A -85,B 0,C 180,E1 -21079.869,E2 -21079.869} C_VEL
LIN {X 0,Y 206.762,Z 413.197,A -85,B 0,C 180,E1 -21084.072,E2 -21084.072} C_VEL
LIN {X 0,Y 206.743,Z 413.229,A -85,B 0,C 180,E1 -21088.419,E2 -21088.419} C_VEL
LIN {X 0,Y 206.701,Z 413.212,A -85,B 0,C 180,E1 -21092.957,E2 -21092.957} C_VEL
LIN {X 0,Y 206.679,Z 413.24,A -85,B 0,C 180,E1 -21097.74,E2 -21097.74} C_VEL
LIN {X 0,Y 206.642,Z 413.223,A -85,B 0,C 180,E1 -21101.563,E2 -21101.563} C_VEL
LIN {X 0,Y 206.677,Z 413.241,A -85,B 0,C 180,E1 -21105.569,E2 -21105.569} C_VEL
LIN {X 0,Y 206.719,Z 413.223,A -85,B 0,C 180,E1 -21109.763,E2 -21109.763} C_VEL
LIN {X 0,Y 206.725,Z 413.237,A -85,B 0,C 180,E1 -21112.27,E2 -21112.27} C_VEL
LIN {X 0,Y 206.709,Z 413.19,A -85,B 0,C 180,E1 -21117.044,E2 -21117.044} C_VEL
LIN {X 0,Y 206.767,Z 413.229,A -85,B 0,C 180,E1 -21122.096,E2 -21122.096} C_VEL
LIN {X 0,Y 206.816,Z 413.334,A -85,B 0,C 180,E1 -21127.627,E2 -21127.627} C_VEL
LIN {X 0,Y 207.015,Z 414.154,A -85,B 0,C 180,E1 -21128.019,E2 -21128.019} C_VEL
LIN {X 0,Y 210.803,Z 422.207,A -85,B 0,C 180,E1 -21128.987,E2 -21128.987} C_VEL
LIN {X 0,Y 217.623,Z 438.68,A -85,B 0,C 180,E1 -21130.587,E2 -21130.587} C_VEL
LIN {X 0,Y 221.674,Z 450.746,A -85,B 0,C 180,E1 -21131.564,E2 -21131.564} C_VEL
LIN {X 0,Y 222.64,Z 458.88,A -85,B 0,C 180,E1 -21131.977,E2 -21131.977} C_VEL
LIN {X 0,Y 220.239,Z 520.291,A -85,B 0,C 180,E1 -21133.905,E2 -21133.905} C_VEL
LIN {X 0,Y 219.181,Z 533.648,A -85,B 0,C 180,E1 -21134.661,E2 -21134.661} C_VEL
LIN {X 0,Y 217.808,Z 545.799,A -85,B 0,C 180,E1 -21135.691,E2 -21135.691} C_VEL
LIN {X 0,Y 216.12,Z 557.779,A -85,B 0,C 180,E1 -21137.081,E2 -21137.081} C_VEL
LIN {X 0,Y 213.973,Z 569.498,A -85,B 0,C 180,E1 -21138.874,E2 -21138.874} C_VEL
LIN {X 0,Y 212.149,Z 578.925,A -85,B 0,C 180,E1 -21140.706,E2 -21140.706} C_VEL
LIN {X 0,Y 210.348,Z 587.685,A -85,B 0,C 180,E1 -21142.802,E2 -21142.802} C_VEL
LIN {X 0,Y 208.71,Z 595.734,A -85,B 0,C 180,E1 -21145.171,E2 -21145.171} C_VEL
LIN {X 0,Y 206.964,Z 603.651,A -85,B 0,C 180,E1 -21148.054,E2 -21148.054} C_VEL
LIN {X 0,Y 205.808,Z 609.951,A -85,B 0,C 180,E1 -21150.978,E2 -21150.978} C_VEL
LIN {X 0,Y 205.023,Z 614.968,A -85,B 0,C 180,E1 -21153.931,E2 -21153.931} C_VEL
LIN {X 0,Y 204.44,Z 618.859,A -85,B 0,C 180,E1 -21156.91,E2 -21156.91} C_VEL
LIN {X 0,Y 204.059,Z 621.716,A -85,B 0,C 180,E1 -21159.915,E2 -21159.915} C_VEL
LIN {X 0,Y 203.981,Z 623.063,A -85,B 0,C 180,E1 -21161.93,E2 -21161.93} C_VEL
LIN {X 0,Y 204.107,Z 624.413,A -85,B 0,C 180,E1 -21165.394,E2 -21165.394} C_VEL
LIN {X 0,Y 204.346,Z 624.619,A -85,B 0,C 180,E1 -21168.03,E2 -21168.03} C_VEL
LIN {X 0,Y 204.719,Z 624.3,A -85,B 0,C 180,E1 -21170.077,E2 -21170.077} C_VEL
LIN {X 0,Y 205.415,Z 623.373,A -85,B 0,C 180,E1 -21172.517,E2 -21172.517} C_VEL
LIN {X 0,Y 206.96,Z 620.751,A -85,B 0,C 180,E1 -21176.196,E2 -21176.196} C_VEL
LIN {X 0,Y 208.49,Z 617.979,A -85,B 0,C 180,E1 -21178.785,E2 -21178.785} C_VEL
LIN {X 0,Y 211.155,Z 612.956,A -85,B 0,C 180,E1 -21182.176,E2 -21182.176} C_VEL
LIN {X 0,Y 214.144,Z 606.896,A -85,B 0,C 180,E1 -21185.215,E2 -21185.215} C_VEL
LIN {X 0,Y 217.412,Z 599.911,A -85,B 0,C 180,E1 -21187.891,E2 -21187.891} C_VEL
LIN {X 0,Y 220.94,Z 591.583,A -85,B 0,C 180,E1 -21190.392,E2 -21190.392} C_VEL
LIN {X 0,Y 224.608,Z 582.262,A -85,B 0,C 180,E1 -21192.581,E2 -21192.581} C_VEL
LIN {X 0,Y 228.103,Z 571.901,A -85,B 0,C 180,E1 -21194.501,E2 -21194.501} C_VEL
LIN {X 0,Y 231.428,Z 560.121,A -85,B 0,C 180,E1 -21196.181,E2 -21196.181} C_VEL
LIN {X 0,Y 233.951,Z 549.138,A -85,B 0,C 180,E1 -21197.389,E2 -21197.389} C_VEL
LIN {X 0,Y 236.191,Z 537.438,A -85,B 0,C 180,E1 -21198.328,E2 -21198.328} C_VEL
LIN {X 0,Y 237.91,Z 524.192,A -85,B 0,C 180,E1 -21199.062,E2 -21199.062} C_VEL
LIN {X 0,Y 239.137,Z 506.184,A -85,B 0,C 180,E1 -21199.643,E2 -21199.643} C_VEL
LIN {X 0,Y 240.943,Z 472.362,A -85,B 0,C 180,E1 -21200.606,E2 -21200.606} C_VEL
LIN {X 0,Y 235.7,Z 460.595,A -85,B 0,C 180,E1 -21202.302,E2 -21202.302} C_VEL
LIN {X 0,Y 230.022,Z 449.647,A -85,B 0,C 180,E1 -21204.219,E2 -21204.219} C_VEL
LIN {X 0,Y 224.018,Z 439.18,A -85,B 0,C 180,E1 -21206.381,E2 -21206.381} C_VEL
LIN {X 0,Y 218.086,Z 430.049,A -85,B 0,C 180,E1 -21208.675,E2 -21208.675} C_VEL
LIN {X 0,Y 214.221,Z 424.566,A -85,B 0,C 180,E1 -21210.28,E2 -21210.28} C_VEL
LIN {X 0,Y 210.621,Z 419.559,A -85,B 0,C 180,E1 -21211.88,E2 -21211.88} C_VEL
LIN {X 0,Y 207.327,Z 415.308,A -85,B 0,C 180,E1 -21213.479,E2 -21213.479} C_VEL
LIN {X 0,Y 206.893,Z 414.055,A -85,B 0,C 180,E1 -21214.065,E2 -21214.065} C_VEL
LIN {X 0,Y 206.767,Z 413.232,A -85,B 0,C 180,E1 -21214.992,E2 -21214.992} C_VEL
LIN {X 0,Y 206.779,Z 413.226,A -85,B 0,C 180,E1 -21220.131,E2 -21220.131} C_VEL
LIN {X 0,Y 206.861,Z 413.212,A -85,B 0,C 180,E1 -21224.229,E2 -21224.229} C_VEL
LIN {X 0,Y 207.092,Z 413.175,A -85,B 0,C 180,E1 -21229.78,E2 -21229.78} C_VEL
LIN {X 0,Y 207.173,Z 413.18,A -85,B 0,C 180,E1 -21232.201,E2 -21232.201} C_VEL
LIN {X 0,Y 207.409,Z 413.138,A -85,B 0,C 180,E1 -21238.058,E2 -21238.058} C_VEL
LIN {X 0,Y 207.514,Z 413.124,A -85,B 0,C 180,E1 -21240,E2 -21240} C_VEL
LIN {X 0,Y 207.379,Z 413.152,A -85,B 0,C 180,E1 -21241.942,E2 -21241.942} C_VEL
LIN {X 0,Y 207.163,Z 413.168,A -85,B 0,C 180,E1 -21247.799,E2 -21247.799} C_VEL
LIN {X 0,Y 206.977,Z 413.201,A -85,B 0,C 180,E1 -21251.756,E2 -21251.756} C_VEL
LIN {X 0,Y 206.863,Z 413.218,A -85,B 0,C 180,E1 -21255.771,E2 -21255.771} C_VEL
LIN {X 0,Y 206.779,Z 413.222,A -85,B 0,C 180,E1 -21259.87,E2 -21259.87} C_VEL
LIN {X 0,Y 206.76,Z 413.224,A -85,B 0,C 180,E1 -21264.073,E2 -21264.073} C_VEL
LIN {X 0,Y 206.74,Z 413.23,A -85,B 0,C 180,E1 -21268.42,E2 -21268.42} C_VEL
LIN {X 0,Y 206.706,Z 413.234,A -85,B 0,C 180,E1 -21272.957,E2 -21272.957} C_VEL
LIN {X 0,Y 206.744,Z 413.396,A -85,B 0,C 180,E1 -21276.051,E2 -21276.051} C_VEL
LIN {X 0,Y 208.146,Z 417.728,A -85,B 0,C 180,E1 -21279.769,E2 -21279.769} C_VEL
LIN {X 0,Y 211.041,Z 422.252,A -85,B 0,C 180,E1 -21281.285,E2 -21281.285} C_VEL
LIN {X 0,Y 213.013,Z 424.92,A -85,B 0,C 180,E1 -21282.161,E2 -21282.161} C_VEL
LIN {X 0,Y 216.678,Z 430.434,A -85,B 0,C 180,E1 -21283.731,E2 -21283.731} C_VEL
LIN {X 0,Y 217.442,Z 431.678,A -85,B 0,C 180,E1 -21284.05,E2 -21284.05} C_VEL
LIN {X 0,Y 219.065,Z 434.206,A -85,B 0,C 180,E1 -21284.708,E2 -21284.708} C_VEL
LIN {X 0,Y 220.371,Z 437.205,A -85,B 0,C 180,E1 -21285.272,E2 -21285.272} C_VEL
LIN {X 0,Y 222.322,Z 443.991,A -85,B 0,C 180,E1 -21286.204,E2 -21286.204} C_VEL
LIN {X 0,Y 225.001,Z 454.719,A -85,B 0,C 180,E1 -21287.498,E2 -21287.498} C_VEL
LIN {X 0,Y 226.24,Z 458.017,A -85,B 0,C 180,E1 -21287.998,E2 -21287.998} C_VEL
LIN {X 0,Y 232.549,Z 471.343,A -85,B 0,C 180,E1 -21290.243,E2 -21290.243} C_VEL
LIN {X 0,Y 235.537,Z 478.451,A -85,B 0,C 180,E1 -21291.266,E2 -21291.266} C_VEL
LIN {X 0,Y 232.711,Z 526.382,A -85,B 0,C 180,E1 -21292.679,E2 -21292.679} C_VEL
LIN {X 0,Y 231.052,Z 539.649,A -85,B 0,C 180,E1 -21293.35,E2 -21293.35} C_VEL
LIN {X 0,Y 228.776,Z 552.105,A -85,B 0,C 180,E1 -21294.292,E2 -21294.292} C_VEL
LIN {X 0,Y 225.975,Z 563.265,A -85,B 0,C 180,E1 -21295.419,E2 -21295.419} C_VEL
LIN {X 0,Y 222.658,Z 574.791,A -85,B 0,C 180,E1 -21297.012,E2 -21297.012} C_VEL
LIN {X 0,Y 219.059,Z 585.189,A -85,B 0,C 180,E1 -21298.848,E2 -21298.848} C_VEL
LIN {X 0,Y 215.67,Z 593.709,A -85,B 0,C 180,E1 -21300.739,E2 -21300.739} C_VEL
LIN {X 0,Y 212.223,Z 601.578,A -85,B 0,C 180,E1 -21302.914,E2 -21302.914} C_VEL
LIN {X 0,Y 208.867,Z 608.929,A -85,B 0,C 180,E1 -21305.488,E2 -21305.488} C_VEL
LIN {X 0,Y 206.096,Z 614.568,A -85,B 0,C 180,E1 -21307.97,E2 -21307.97} C_VEL
LIN {X 0,Y 203.299,Z 619.729,A -85,B 0,C 180,E1 -21310.828,E2 -21310.828} C_VEL
LIN {X 0,Y 201.037,Z 623.749,A -85,B 0,C 180,E1 -21313.76,E2 -21313.76} C_VEL
LIN {X 0,Y 199.937,Z 625.847,A -85,B 0,C 180,E1 -21315.757,E2 -21315.757} C_VEL
LIN {X 0,Y 198.261,Z 628.79,A -85,B 0,C 180,E1 -21319.792,E2 -21319.792} C_VEL
LIN {X 0,Y 197.727,Z 629.68,A -85,B 0,C 180,E1 -21321.827,E2 -21321.827} C_VEL
LIN {X 0,Y 197.415,Z 630.15,A -85,B 0,C 180,E1 -21323.87,E2 -21323.87} C_VEL
LIN {X 0,Y 197.24,Z 630.21,A -85,B 0,C 180,E1 -21326.107,E2 -21326.107} C_VEL
LIN {X 0,Y 197.266,Z 629.23,A -85,B 0,C 180,E1 -21330.001,E2 -21330.001} C_VEL
LIN {X 0,Y 197.18,Z 626.965,A -85,B 0,C 180,E1 -21333.629,E2 -21333.629} C_VEL
LIN {X 0,Y 197.434,Z 623.426,A -85,B 0,C 180,E1 -21337.157,E2 -21337.157} C_VEL
LIN {X 0,Y 198.024,Z 619.209,A -85,B 0,C 180,E1 -21340.222,E2 -21340.222} C_VEL
LIN {X 0,Y 199.139,Z 612.767,A -85,B 0,C 180,E1 -21343.782,E2 -21343.782} C_VEL
LIN {X 0,Y 200.681,Z 605.722,A -85,B 0,C 180,E1 -21346.794,E2 -21346.794} C_VEL
LIN {X 0,Y 202.314,Z 598.512,A -85,B 0,C 180,E1 -21349.27,E2 -21349.27} C_VEL
LIN {X 0,Y 204.225,Z 589.257,A -85,B 0,C 180,E1 -21351.841,E2 -21351.841} C_VEL
LIN {X 0,Y 206.362,Z 578.922,A -85,B 0,C 180,E1 -21354.122,E2 -21354.122} C_VEL
LIN {X 0,Y 208.431,Z 568.138,A -85,B 0,C 180,E1 -21355.998,E2 -21355.998} C_VEL
LIN {X 0,Y 210.507,Z 556.031,A -85,B 0,C 180,E1 -21357.596,E2 -21357.596} C_VEL
LIN {X 0,Y 212.15,Z 543.358,A -85,B 0,C 180,E1 -21358.843,E2 -21358.843} C_VEL
LIN {X 0,Y 213.429,Z 530.556,A -85,B 0,C 180,E1 -21359.699,E2 -21359.699} C_VEL
LIN {X 0,Y 214.214,Z 514.525,A -85,B 0,C 180,E1 -21360.326,E2 -21360.326} C_VEL
LIN {X 0,Y 215.874,Z 468.235,A -85,B 0,C 180,E1 -21361.814,E2 -21361.814} C_VEL
LIN {X 0,Y 213.603,Z 450.54,A -85,B 0,C 180,E1 -21362.783,E2 -21362.783} C_VEL
LIN {X 0,Y 208.743,Z 437.258,A -85,B 0,C 180,E1 -21363.995,E2 -21363.995} C_VEL
LIN {X 0,Y 202.154,Z 421.752,A -85,B 0,C 180,E1 -21365.644,E2 -21365.644} C_VEL
LIN {X 0,Y 200.68,Z 418.281,A -85,B 0,C 180,E1 -21366.131,E2 -21366.131} C_VEL
LIN {X 0,Y 199.67,Z 414.179,A -85,B 0,C 180,E1 -21368.343,E2 -21368.343} C_VEL
LIN {X 0,Y 199.63,Z 414.115,A -85,B 0,C 180,E1 -21372.327,E2 -21372.327} C_VEL
LIN {X 0,Y 199.665,Z 414.065,A -85,B 0,C 180,E1 -21375.252,E2 -21375.252} C_VEL
LIN {X 0,Y 199.665,Z 414.079,A -85,B 0,C 180,E1 -21378.027,E2 -21378.027} C_VEL
LIN {X 0,Y 199.68,Z 414.112,A -85,B 0,C 180,E1 -21380.743,E2 -21380.743} C_VEL
LIN {X 0,Y 199.633,Z 414.11,A -85,B 0,C 180,E1 -21385.717,E2 -21385.717} C_VEL
LIN {X 0,Y 199.696,Z 414.111,A -85,B 0,C 180,E1 -21388.136,E2 -21388.136} C_VEL
LIN {X 0,Y 199.684,Z 414.1,A -85,B 0,C 180,E1 -21392.771,E2 -21392.771} C_VEL
LIN {X 0,Y 199.713,Z 414.099,A -85,B 0,C 180,E1 -21397.226,E2 -21397.226} C_VEL
LIN {X 0,Y 199.794,Z 414.083,A -85,B 0,C 180,E1 -21401.758,E2 -21401.758} C_VEL
LIN {X 0,Y 199.833,Z 414.089,A -85,B 0,C 180,E1 -21405.748,E2 -21405.748} C_VEL
LIN {X 0,Y 200.021,Z 414.036,A -85,B 0,C 180,E1 -21409.881,E2 -21409.881} C_VEL
LIN {X 0,Y 200.021,Z 414.068,A -85,B 0,C 180,E1 -21413.949,E2 -21413.949} C_VEL
LIN {X 0,Y 200.319,Z 414.02,A -85,B 0,C 180,E1 -21417.989,E2 -21417.989} C_VEL
LIN {X 0,Y 200.477,Z 413.979,A -85,B 0,C 180,E1 -21420,E2 -21420} C_VEL
LIN {X 0,Y 200.026,Z 414.057,A -85,B 0,C 180,E1 -21424.029,E2 -21424.029} C_VEL
LIN {X 0,Y 200.093,Z 414.057,A -85,B 0,C 180,E1 -21428.076,E2 -21428.076} C_VEL
LIN {X 0,Y 199.872,Z 414.05,A -85,B 0,C 180,E1 -21432.179,E2 -21432.179} C_VEL
LIN {X 0,Y 199.802,Z 414.091,A -85,B 0,C 180,E1 -21436.344,E2 -21436.344} C_VEL
LIN {X 0,Y 199.698,Z 414.099,A -85,B 0,C 180,E1 -21440.605,E2 -21440.605} C_VEL
LIN {X 0,Y 199.672,Z 414.085,A -85,B 0,C 180,E1 -21444.984,E2 -21444.984} C_VEL
LIN {X 0,Y 199.674,Z 414.11,A -85,B 0,C 180,E1 -21449.522,E2 -21449.522} C_VEL
LIN {X 0,Y 199.676,Z 414.089,A -85,B 0,C 180,E1 -21452.358,E2 -21452.358} C_VEL
LIN {X 0,Y 199.622,Z 414.114,A -85,B 0,C 180,E1 -21456.763,E2 -21456.763} C_VEL
LIN {X 0,Y 199.608,Z 414.117,A -85,B 0,C 180,E1 -21459.328,E2 -21459.328} C_VEL
LIN {X 0,Y 199.574,Z 414.102,A -85,B 0,C 180,E1 -21462.311,E2 -21462.311} C_VEL
LIN {X 0,Y 199.612,Z 414.121,A -85,B 0,C 180,E1 -21465.238,E2 -21465.238} C_VEL
LIN {X 0,Y 199.649,Z 414.105,A -85,B 0,C 180,E1 -21468.023,E2 -21468.023} C_VEL
LIN {X 0,Y 199.679,Z 414.108,A -85,B 0,C 180,E1 -21470.744,E2 -21470.744} C_VEL
LIN {X 0,Y 199.634,Z 414.079,A -85,B 0,C 180,E1 -21475.718,E2 -21475.718} C_VEL
LIN {X 0,Y 199.704,Z 414.062,A -85,B 0,C 180,E1 -21478.138,E2 -21478.138} C_VEL
LIN {X 0,Y 199.687,Z 414.099,A -85,B 0,C 180,E1 -21482.772,E2 -21482.772} C_VEL
LIN {X 0,Y 199.76,Z 414.239,A -85,B 0,C 180,E1 -21486.546,E2 -21486.546} C_VEL
LIN {X 0,Y 200.032,Z 415.343,A -85,B 0,C 180,E1 -21486.961,E2 -21486.961} C_VEL
LIN {X 0,Y 204.842,Z 424.819,A -85,B 0,C 180,E1 -21488.167,E2 -21488.167} C_VEL
LIN {X 0,Y 211.72,Z 441.544,A -85,B 0,C 180,E1 -21489.863,E2 -21489.863} C_VEL
LIN {X 0,Y 215.538,Z 453.134,A -85,B 0,C 180,E1 -21490.837,E2 -21490.837} C_VEL
LIN {X 0,Y 216.273,Z 459.216,A -85,B 0,C 180,E1 -21491.161,E2 -21491.161} C_VEL
LIN {X 0,Y 213.749,Z 520.927,A -85,B 0,C 180,E1 -21493.157,E2 -21493.157} C_VEL
LIN {X 0,Y 212.656,Z 534.094,A -85,B 0,C 180,E1 -21493.932,E2 -21493.932} C_VEL
LIN {X 0,Y 211.11,Z 547.214,A -85,B 0,C 180,E1 -21495.097,E2 -21495.097} C_VEL
LIN {X 0,Y 209.214,Z 559.648,A -85,B 0,C 180,E1 -21496.647,E2 -21496.647} C_VEL
LIN {X 0,Y 207.031,Z 571.035,A -85,B 0,C 180,E1 -21498.496,E2 -21498.496} C_VEL
LIN {X 0,Y 205.188,Z 580.212,A -85,B 0,C 180,E1 -21500.388,E2 -21500.388} C_VEL
LIN {X 0,Y 203.277,Z 588.785,A -85,B 0,C 180,E1 -21502.55,E2 -21502.55} C_VEL
LIN {X 0,Y 201.625,Z 596.664,A -85,B 0,C 180,E1 -21505,E2 -21505} C_VEL
LIN {X 0,Y 199.855,Z 604.379,A -85,B 0,C 180,E1 -21507.984,E2 -21507.984} C_VEL
LIN {X 0,Y 198.666,Z 610.56,A -85,B 0,C 180,E1 -21511.013,E2 -21511.013} C_VEL
LIN {X 0,Y 197.879,Z 615.47,A -85,B 0,C 180,E1 -21514.073,E2 -21514.073} C_VEL
LIN {X 0,Y 197.292,Z 619.263,A -85,B 0,C 180,E1 -21517.161,E2 -21517.161} C_VEL
LIN {X 0,Y 196.938,Z 622.024,A -85,B 0,C 180,E1 -21520.278,E2 -21520.278} C_VEL
LIN {X 0,Y 196.871,Z 623.327,A -85,B 0,C 180,E1 -21522.367,E2 -21522.367} C_VEL
LIN {X 0,Y 197.022,Z 624.502,A -85,B 0,C 180,E1 -21525.609,E2 -21525.609} C_VEL
LIN {X 0,Y 197.345,Z 624.7,A -85,B 0,C 180,E1 -21528.693,E2 -21528.693} C_VEL
LIN {X 0,Y 197.795,Z 624.334,A -85,B 0,C 180,E1 -21530.812,E2 -21530.812} C_VEL
LIN {X 0,Y 198.438,Z 623.522,A -85,B 0,C 180,E1 -21532.952,E2 -21532.952} C_VEL
LIN {X 0,Y 199.256,Z 622.277,A -85,B 0,C 180,E1 -21535.039,E2 -21535.039} C_VEL
LIN {X 0,Y 200.938,Z 619.568,A -85,B 0,C 180,E1 -21538.174,E2 -21538.174} C_VEL
LIN {X 0,Y 203.149,Z 615.767,A -85,B 0,C 180,E1 -21541.259,E2 -21541.259} C_VEL
LIN {X 0,Y 205.874,Z 610.758,A -85,B 0,C 180,E1 -21544.281,E2 -21544.281} C_VEL
LIN {X 0,Y 209.121,Z 604.386,A -85,B 0,C 180,E1 -21547.222,E2 -21547.222} C_VEL
LIN {X 0,Y 212.932,Z 596.358,A -85,B 0,C 180,E1 -21550.06,E2 -21550.06} C_VEL
LIN {X 0,Y 216.859,Z 587.25,A -85,B 0,C 180,E1 -21552.539,E2 -21552.539} C_VEL
LIN {X 0,Y 220.807,Z 576.782,A -85,B 0,C 180,E1 -21554.764,E2 -21554.764} C_VEL
LIN {X 0,Y 224.447,Z 565.474,A -85,B 0,C 180,E1 -21556.594,E2 -21556.594} C_VEL
LIN {X 0,Y 227.644,Z 553.124,A -85,B 0,C 180,E1 -21558.14,E2 -21558.14} C_VEL
LIN {X 0,Y 230.25,Z 540.871,A -85,B 0,C 180,E1 -21559.23,E2 -21559.23} C_VEL
LIN {X 0,Y 232.238,Z 527.935,A -85,B 0,C 180,E1 -21560.037,E2 -21560.037} C_VEL
LIN {X 0,Y 233.489,Z 514.468,A -85,B 0,C 180,E1 -21560.556,E2 -21560.556} C_VEL
LIN {X 0,Y 235.721,Z 474.799,A -85,B 0,C 180,E1 -21561.696,E2 -21561.696} C_VEL
LIN {X 0,Y 230.477,Z 463.041,A -85,B 0,C 180,E1 -21563.498,E2 -21563.498} C_VEL
LIN {X 0,Y 224.118,Z 450.857,A -85,B 0,C 180,E1 -21565.789,E2 -21565.789} C_VEL
LIN {X 0,Y 217.936,Z 440.3,A -85,B 0,C 180,E1 -21568.19,E2 -21568.19} C_VEL
LIN {X 0,Y 211.306,Z 430.467,A -85,B 0,C 180,E1 -21570.996,E2 -21570.996} C_VEL
LIN {X 0,Y 207.679,Z 425.347,A -85,B 0,C 180,E1 -21572.683,E2 -21572.683} C_VEL
LIN {X 0,Y 204.281,Z 420.827,A -85,B 0,C 180,E1 -21574.393,E2 -21574.393} C_VEL
LIN {X 0,Y 202.819,Z 419.139,A -85,B 0,C 180,E1 -21575.156,E2 -21575.156} C_VEL
LIN {X 0,Y 200.736,Z 416.974,A -85,B 0,C 180,E1 -21576.275,E2 -21576.275} C_VEL
LIN {X 0,Y 199.783,Z 414.492,A -85,B 0,C 180,E1 -21577.132,E2 -21577.132} C_VEL
LIN {X 0,Y 199.721,Z 414.111,A -85,B 0,C 180,E1 -21577.773,E2 -21577.773} C_VEL
LIN {X 0,Y 199.792,Z 414.087,A -85,B 0,C 180,E1 -21581.757,E2 -21581.757} C_VEL
LIN {X 0,Y 199.842,Z 414.079,A -85,B 0,C 180,E1 -21585.749,E2 -21585.749} C_VEL
LIN {X 0,Y 200.066,Z 414.05,A -85,B 0,C 180,E1 -21589.884,E2 -21589.884} C_VEL
LIN {X 0,Y 200.036,Z 414.053,A -85,B 0,C 180,E1 -21593.95,E2 -21593.95} C_VEL
LIN {X 0,Y 200.345,Z 414.018,A -85,B 0,C 180,E1 -21597.99,E2 -21597.99} C_VEL
LIN {X 0,Y 200.478,Z 414,A -85,B 0,C 180,E1 -21600,E2 -21600} C_VEL
LIN {X 0,Y 200.028,Z 414.052,A -85,B 0,C 180,E1 -21604.03,E2 -21604.03} C_VEL
LIN {X 0,Y 200.106,Z 414.045,A -85,B 0,C 180,E1 -21608.076,E2 -21608.076} C_VEL
LIN {X 0,Y 199.909,Z 414.076,A -85,B 0,C 180,E1 -21612.177,E2 -21612.177} C_VEL
LIN {X 0,Y 199.8,Z 414.096,A -85,B 0,C 180,E1 -21616.344,E2 -21616.344} C_VEL
LIN {X 0,Y 199.695,Z 414.111,A -85,B 0,C 180,E1 -21620.606,E2 -21620.606} C_VEL
LIN {X 0,Y 199.669,Z 414.113,A -85,B 0,C 180,E1 -21624.985,E2 -21624.985} C_VEL
LIN {X 0,Y 199.671,Z 414.107,A -85,B 0,C 180,E1 -21629.523,E2 -21629.523} C_VEL
LIN {X 0,Y 199.685,Z 414.194,A -85,B 0,C 180,E1 -21633.215,E2 -21633.215} C_VEL
LIN {X 0,Y 200.678,Z 417.38,A -85,B 0,C 180,E1 -21636.405,E2 -21636.405} C_VEL
LIN {X 0,Y 203.426,Z 421.68,A -85,B 0,C 180,E1 -21638.138,E2 -21638.138} C_VEL
LIN {X 0,Y 205.631,Z 424.401,A -85,B 0,C 180,E1 -21639.268,E2 -21639.268} C_VEL
LIN {X 0,Y 209.874,Z 430.525,A -85,B 0,C 180,E1 -21641.325,E2 -21641.325} C_VEL
LIN {X 0,Y 213.741,Z 436.484,A -85,B 0,C 180,E1 -21643.058,E2 -21643.058} C_VEL
LIN {X 0,Y 217.453,Z 442.416,A -85,B 0,C 180,E1 -21644.615,E2 -21644.615} C_VEL
LIN {X 0,Y 221.863,Z 449.832,A -85,B 0,C 180,E1 -21646.355,E2 -21646.355} C_VEL
LIN {X 0,Y 226.24,Z 458.017,A -85,B 0,C 180,E1 -21647.998,E2 -21647.998} C_VEL
LIN {X 0,Y 227.991,Z 462.976,A -85,B 0,C 180,E1 -21648.7,E2 -21648.7} C_VEL
LIN {X 0,Y 229.17,Z 468.386,A -85,B 0,C 180,E1 -21649.256,E2 -21649.256} C_VEL
LIN {X 0,Y 229.986,Z 476.037,A -85,B 0,C 180,E1 -21649.807,E2 -21649.807} C_VEL
LIN {X 0,Y 230.124,Z 479.975,A -85,B 0,C 180,E1 -21650.016,E2 -21650.016} C_VEL
LIN {X 0,Y 229.964,Z 487.939,A -85,B 0,C 180,E1 -21650.327,E2 -21650.327} C_VEL
LIN {X 0,Y 227.463,Z 526.98,A -85,B 0,C 180,E1 -21651.498,E2 -21651.498} C_VEL
LIN {X 0,Y 225.699,Z 540.281,A -85,B 0,C 180,E1 -21652.192,E2 -21652.192} C_VEL
LIN {X 0,Y 223.335,Z 552.534,A -85,B 0,C 180,E1 -21653.141,E2 -21653.141} C_VEL
LIN {X 0,Y 220.216,Z 564.332,A -85,B 0,C 180,E1 -21654.38,E2 -21654.38} C_VEL
LIN {X 0,Y 216.792,Z 575.643,A -85,B 0,C 180,E1 -21656,E2 -21656} C_VEL
LIN {X 0,Y 213.054,Z 585.88,A -85,B 0,C 180,E1 -21657.866,E2 -21657.866} C_VEL
LIN {X 0,Y 209.543,Z 594.267,A -85,B 0,C 180,E1 -21659.796,E2 -21659.796} C_VEL
LIN {X 0,Y 205.945,Z 602.024,A -85,B 0,C 180,E1 -21662.017,E2 -21662.017} C_VEL
LIN {X 0,Y 202.252,Z 609.609,A -85,B 0,C 180,E1 -21664.807,E2 -21664.807} C_VEL
LIN {X 0,Y 198.52,Z 616.632,A -85,B 0,C 180,E1 -21668.179,E2 -21668.179} C_VEL
LIN {X 0,Y 195.767,Z 621.324,A -85,B 0,C 180,E1 -21671.151,E2 -21671.151} C_VEL
LIN {X 0,Y 193.613,Z 624.927,A -85,B 0,C 180,E1 -21674.203,E2 -21674.203} C_VEL
LIN {X 0,Y 192.044,Z 627.545,A -85,B 0,C 180,E1 -21677.317,E2 -21677.317} C_VEL
LIN {X 0,Y 190.702,Z 629.639,A -85,B 0,C 180,E1 -21681.524,E2 -21681.524} C_VEL
LIN {X 0,Y 190.166,Z 630.109,A -85,B 0,C 180,E1 -21685.762,E2 -21685.762} C_VEL
LIN {X 0,Y 190.101,Z 629.774,A -85,B 0,C 180,E1 -21687.882,E2 -21687.882} C_VEL
LIN {X 0,Y 190.173,Z 629.054,A -85,B 0,C 180,E1 -21690.001,E2 -21690.001} C_VEL
LIN {X 0,Y 190.09,Z 627.008,A -85,B 0,C 180,E1 -21693.393,E2 -21693.393} C_VEL
LIN {X 0,Y 190.278,Z 624.295,A -85,B 0,C 180,E1 -21696.362,E2 -21696.362} C_VEL
LIN {X 0,Y 190.757,Z 620.382,A -85,B 0,C 180,E1 -21699.544,E2 -21699.544} C_VEL
LIN {X 0,Y 191.64,Z 615.316,A -85,B 0,C 180,E1 -21702.711,E2 -21702.711} C_VEL
LIN {X 0,Y 192.96,Z 608.922,A -85,B 0,C 180,E1 -21705.853,E2 -21705.853} C_VEL
LIN {X 0,Y 194.793,Z 600.892,A -85,B 0,C 180,E1 -21708.948,E2 -21708.948} C_VEL
LIN {X 0,Y 196.557,Z 593.464,A -85,B 0,C 180,E1 -21711.266,E2 -21711.266} C_VEL
LIN {X 0,Y 198.609,Z 583.742,A -85,B 0,C 180,E1 -21713.736,E2 -21713.736} C_VEL
LIN {X 0,Y 200.902,Z 572.767,A -85,B 0,C 180,E1 -21715.93,E2 -21715.93} C_VEL
LIN {X 0,Y 202.984,Z 562.012,A -85,B 0,C 180,E1 -21717.586,E2 -21717.586} C_VEL
LIN {X 0,Y 204.938,Z 549.006,A -85,B 0,C 180,E1 -21719.113,E2 -21719.113} C_VEL
LIN {X 0,Y 206.397,Z 536.608,A -85,B 0,C 180,E1 -21720.149,E2 -21720.149} C_VEL
LIN {X 0,Y 207.441,Z 523.352,A -85,B 0,C 180,E1 -21720.848,E2 -21720.848} C_VEL
LIN {X 0,Y 209.529,Z 468.836,A -85,B 0,C 180,E1 -21722.664,E2 -21722.664} C_VEL
LIN {X 0,Y 207.44,Z 452.557,A -85,B 0,C 180,E1 -21723.595,E2 -21723.595} C_VEL
LIN {X 0,Y 201.966,Z 437.812,A -85,B 0,C 180,E1 -21725.027,E2 -21725.027} C_VEL
LIN {X 0,Y 196.456,Z 424.964,A -85,B 0,C 180,E1 -21726.481,E2 -21726.481} C_VEL
LIN {X 0,Y 193.416,Z 418.272,A -85,B 0,C 180,E1 -21727.403,E2 -21727.403} C_VEL
LIN {X 0,Y 192.63,Z 415.053,A -85,B 0,C 180,E1 -21729.237,E2 -21729.237} C_VEL
LIN {X 0,Y 192.575,Z 414.96,A -85,B 0,C 180,E1 -21733.9,E2 -21733.9} C_VEL
LIN {X 0,Y 192.604,Z 414.943,A -85,B 0,C 180,E1 -21736.868,E2 -21736.868} C_VEL
LIN {X 0,Y 192.601,Z 414.994,A -85,B 0,C 180,E1 -21741.659,E2 -21741.659} C_VEL
LIN {X 0,Y 192.598,Z 414.995,A -85,B 0,C 180,E1 -21746.814,E2 -21746.814} C_VEL
LIN {X 0,Y 192.66,Z 414.966,A -85,B 0,C 180,E1 -21751.691,E2 -21751.691} C_VEL
LIN {X 0,Y 192.684,Z 414.982,A -85,B 0,C 180,E1 -21756.345,E2 -21756.345} C_VEL
LIN {X 0,Y 192.73,Z 414.959,A -85,B 0,C 180,E1 -21761.459,E2 -21761.459} C_VEL
LIN {X 0,Y 192.761,Z 414.973,A -85,B 0,C 180,E1 -21765.213,E2 -21765.213} C_VEL
LIN {X 0,Y 192.944,Z 414.916,A -85,B 0,C 180,E1 -21769.566,E2 -21769.566} C_VEL
LIN {X 0,Y 192.983,Z 414.943,A -85,B 0,C 180,E1 -21773.728,E2 -21773.728} C_VEL
LIN {X 0,Y 193.261,Z 414.899,A -85,B 0,C 180,E1 -21777.916,E2 -21777.916} C_VEL
LIN {X 0,Y 193.441,Z 414.853,A -85,B 0,C 180,E1 -21780,E2 -21780} C_VEL
LIN {X 0,Y 192.972,Z 414.937,A -85,B 0,C 180,E1 -21784.177,E2 -21784.177} C_VEL
LIN {X 0,Y 193.039,Z 414.935,A -85,B 0,C 180,E1 -21788.373,E2 -21788.373} C_VEL
LIN {X 0,Y 192.799,Z 414.929,A -85,B 0,C 180,E1 -21792.633,E2 -21792.633} C_VEL
LIN {X 0,Y 192.756,Z 414.97,A -85,B 0,C 180,E1 -21796.959,E2 -21796.959} C_VEL
LIN {X 0,Y 192.635,Z 414.971,A -85,B 0,C 180,E1 -21801.397,E2 -21801.397} C_VEL
LIN {X 0,Y 192.663,Z 414.951,A -85,B 0,C 180,E1 -21804.224,E2 -21804.224} C_VEL
LIN {X 0,Y 192.649,Z 414.987,A -85,B 0,C 180,E1 -21808.892,E2 -21808.892} C_VEL
LIN {X 0,Y 192.598,Z 414.965,A -85,B 0,C 180,E1 -21813.186,E2 -21813.186} C_VEL
LIN {X 0,Y 192.551,Z 415,A -85,B 0,C 180,E1 -21818.352,E2 -21818.352} C_VEL
LIN {X 0,Y 192.516,Z 414.984,A -85,B 0,C 180,E1 -21823.104,E2 -21823.104} C_VEL
LIN {X 0,Y 192.559,Z 414.996,A -85,B 0,C 180,E1 -21826.883,E2 -21826.883} C_VEL
LIN {X 0,Y 192.6,Z 414.997,A -85,B 0,C 180,E1 -21831.66,E2 -21831.66} C_VEL
LIN {X 0,Y 192.6,Z 414.943,A -85,B 0,C 180,E1 -21836.815,E2 -21836.815} C_VEL
LIN {X 0,Y 192.665,Z 414.987,A -85,B 0,C 180,E1 -21841.692,E2 -21841.692} C_VEL
LIN {X 0,Y 192.678,Z 415.152,A -85,B 0,C 180,E1 -21845.342,E2 -21845.342} C_VEL
LIN {X 0,Y 192.975,Z 416.325,A -85,B 0,C 180,E1 -21845.754,E2 -21845.754} C_VEL
LIN {X 0,Y 198.527,Z 426.743,A -85,B 0,C 180,E1 -21847.203,E2 -21847.203} C_VEL
LIN {X 0,Y 204.909,Z 441.917,A -85,B 0,C 180,E1 -21848.859,E2 -21848.859} C_VEL
LIN {X 0,Y 209.363,Z 455.022,A -85,B 0,C 180,E1 -21850.037,E2 -21850.037} C_VEL
LIN {X 0,Y 209.953,Z 460.053,A -85,B 0,C 180,E1 -21850.316,E2 -21850.316} C_VEL
LIN {X 0,Y 207.298,Z 521.545,A -85,B 0,C 180,E1 -21852.362,E2 -21852.362} C_VEL
LIN {X 0,Y 206.166,Z 534.54,A -85,B 0,C 180,E1 -21853.156,E2 -21853.156} C_VEL
LIN {X 0,Y 204.591,Z 547.302,A -85,B 0,C 180,E1 -21854.324,E2 -21854.324} C_VEL
LIN {X 0,Y 202.853,Z 558.45,A -85,B 0,C 180,E1 -21855.726,E2 -21855.726} C_VEL
LIN {X 0,Y 200.574,Z 569.991,A -85,B 0,C 180,E1 -21857.607,E2 -21857.607} C_VEL
LIN {X 0,Y 198.598,Z 579.37,A -85,B 0,C 180,E1 -21859.551,E2 -21859.551} C_VEL
LIN {X 0,Y 196.641,Z 588.091,A -85,B 0,C 180,E1 -21861.78,E2 -21861.78} C_VEL
LIN {X 0,Y 194.866,Z 596.105,A -85,B 0,C 180,E1 -21864.308,E2 -21864.308} C_VEL
LIN {X 0,Y 192.988,Z 603.982,A -85,B 0,C 180,E1 -21867.39,E2 -21867.39} C_VEL
LIN {X 0,Y 191.932,Z 609.316,A -85,B 0,C 180,E1 -21869.999,E2 -21869.999} C_VEL
